(* IEC 61131-3 sources: HMITools/src/Ar/HMITools, 32 files *)

(* ---- EditorControl.typ ---- *)
(*
* File: EditorControl.typ
* Copyright (c) 2023 Loupe
* https://loupe.team
*
* This file is part of HMITools, licensed under the MIT License.
*
*)
(*Application Editor*)

TYPE
	HMI_Editor_Controller_typ : 	STRUCT
		CMD : HMI_Editor_Controller_CMD_typ;
		HMI : HMI_EditControl_typ;
		Internal : HMI_Editor_Controller_int_typ;
	END_STRUCT;
	HMI_Editor_Controller_int_typ : 	STRUCT
		CMD : HMI_Editor_Controller_CMD_typ;
	END_STRUCT;
	HMI_Editor_Controller_CMD_typ : 	STRUCT
		Load : BOOL;
		Save : BOOL;
		Clear : BOOL;
	END_STRUCT;
END_TYPE

(*HMI Connections*)

TYPE
	HMI_EditControl_Internal_typ : 	STRUCT
		CurrentLineText : STRING[200];
		CurrentLineIndex : UINT;
		CommandState : USINT;
		EditText : STRING[80];
		DesiredLine : USINT;
		DesiredColumn : USINT;
		Offset : USINT;
		Count : USINT;
		highlightmode : USINT;
	END_STRUCT;
	HMI_EditControl_Runtime_Edit_typ : 	STRUCT
		CursorLineDp : UINT;
		CursorColumnDp : UINT;
		InsertModeDp : UINT;
		ModifiedDp : UINT;
		SelectionModeDp : UINT;
	END_STRUCT;
	HMI_EditControl_Runtime_Comp_typ : 	STRUCT
		CompletionDP : UINT;
	END_STRUCT;
	HMI_EditControl_Runtime_Cmds_typ : 	STRUCT
		ResponseDp : STRING[80];
		RequestDp : STRING[80];
		StatusDP : UINT;
	END_STRUCT;
	HMI_EditControl_Runtime_typ : 	STRUCT
		StatusDp : UINT;
		BusyDp : UINT;
		Commands : HMI_EditControl_Runtime_Cmds_typ;
		Completion : HMI_EditControl_Runtime_Comp_typ;
		Edit : HMI_EditControl_Runtime_Edit_typ;
	END_STRUCT;
	HMI_EditControl_Value_typ : 	STRUCT
		Content : STRING[1000];
		URLDp : STRING[80];
	END_STRUCT;
	HMI_EditControl_typ : 	STRUCT
		Value : HMI_EditControl_Value_typ;
		Runtime : HMI_EditControl_Runtime_typ;
		internal : HMI_EditControl_Internal_typ;
		Command : HMI_EditControl_CMDS;
	END_STRUCT;
	HMI_EditControl_CMDS :
		(
		EC_,
		EC_APPEND,
		EC_CLEAR,
		EC_DELETE,
		EC_GET_LINE,
		EC_GET_MARKED_TEXT,
		EC_GET_TEXT_SIZE,
		EC_GOTO,
		EC_HIGHLIGHT,
		EC_INSERT,
		EC_LOAD,
		EC_READ,
		EC_REPLACE_MARKED_TEXT,
		EC_SAVE,
		EC_UPDATE
		);
END_TYPE

(* ---- HMI_Basic.typ ---- *)
(*
* File: HMI_Basic.typ
* Copyright (c) 2023 Loupe
* https://loupe.team
*
* This file is part of HMITools, licensed under the MIT License.
*
*)

TYPE
	HMI_StatusBits_enum :
		(
		HMI_STATBIT_VIS := 0,
		HMI_STATBIT_LOCK,
		HMI_STATBIT_FOCUS,
		HMI_STATBIT_TOUCHPAD
		);
	HMI_Layer_typ : 	STRUCT
		StatusDP : UINT;
	END_STRUCT;
	HMI_Shape_typ : 	STRUCT
		StatusDP : UINT;
		ColorDP : UINT;
	END_STRUCT;
	HMI_Scale_typ : 	STRUCT
		Value : REAL;
		MinDP : REAL;
		MaxDP : REAL;
		RangeStartDP : REAL;
		RangeEndDP : REAL;
		RangeColorDP : UINT;
		StatusDP : UINT;
		ColorDP : UINT;
	END_STRUCT;
	HMI_Listbox_typ : 	STRUCT
		IndexDP : DINT;
		MinDP : UINT;
		MaxDP : UINT;
		OptionDP : UINT;
		StatusDP : UINT;
		ColorDP : UINT;
		CompletionDP : UINT;
		PageSize : UINT;
	END_STRUCT;
	HMI_Bitmap_typ : 	STRUCT
		IndexDP : UINT;
		StatusDP : UINT;
	END_STRUCT;
	HMI_StringIn_typ : 	STRUCT
		String : STRING[HMI_STRLEN_IN];
		StatusDP : UINT;
		ColorDP : UINT;
		CompletionDP : UINT;
	END_STRUCT;
	HMI_Dropdown_typ : 	STRUCT
		IndexDP : UINT;
		StatusDP : UINT;
		ColorDP : UINT;
	END_STRUCT;
	HMI_TextBox_typ : 	STRUCT
		IndexDP : UINT;
		StatusDP : UINT;
		ColorDP : UINT;
	END_STRUCT;
	HMI_NumericIn_typ : 	STRUCT
		Value : REAL;
		MinDP : REAL;
		MaxDP : REAL;
		StatusDP : UINT;
		ColorDP : UINT;
		CompletionDP : UINT;
	END_STRUCT;
	HMI_NumericOut_typ : 	STRUCT
		Value : REAL;
		StatusDP : UINT;
		ColorDP : UINT;
	END_STRUCT;
	HMI_ButtonVC3_typ : 	STRUCT
		CMD : USINT;
		Lock : UINT;
		ColorDP : UINT;
		LEDDP : USINT;
	END_STRUCT;
	HMI_Button_typ : 	STRUCT
		CMD : BOOL;
		Confirm : BOOL;
		StatusDP : UINT;
		IndexDP : UINT;
		ColorDP : UINT;
		LEDDP : USINT;
	END_STRUCT;
	HMI_SecondaryTab_typ : 	STRUCT
		ChangeToSecondaryTab : BOOL; (*CMD to change to this secondary tab*)
		PageIndex : UINT; (*Page index for this secondary tab*)
	END_STRUCT;
	HMI_PrimaryTab_typ : 	STRUCT
		CurrentSecondaryTab : UINT; (*Current secondary tab*)
		ChangeToPrimaryTab : BOOL; (*CMD to change to this primary tab*)
		Group : UINT; (*Group to which the primary tab belongs*)
		SecondaryTabArray : ARRAY[0..HMI_MAI_TABS]OF HMI_SecondaryTab_typ; (*Array of secondary tabs*)
	END_STRUCT;
	HMI_Tabs_typ : 	STRUCT
		CurrentPrimaryTab : UINT;
		PrimaryTabArray : ARRAY[0..HMI_MAI_TABS]OF HMI_PrimaryTab_typ;
	END_STRUCT;
	HMI_Basic_typ : 	STRUCT
		PageChangeDP : UINT;
		PageCurrentDP : UINT;
		LanguageChangeDP : UINT;
		LanguageCurrentDP : UINT;
		ScreensaverDP : UINT;
		ScreensaverTimeDP : UINT;
		BacklightDP : UINT;
		BacklightTimeDP : UINT;
		CalibrationStateDP : UINT;
		VCHandle : UDINT;
		Tabs : HMI_Tabs_typ;
	END_STRUCT;
END_TYPE

(* ---- HMI_File_Browse.typ ---- *)
(*
* File: HMI_File_Browse.typ
* Copyright (c) 2023 Loupe
* https://loupe.team
*
* This file is part of HMITools, licensed under the MIT License.
*
*)

TYPE
	HMI_File_Browse_internal_typ : 	STRUCT
		TempFileList : UDINT;
		TempFileSelection : STRING[LIST_BOX_STRING_SIZE];
		oldFileIndex : DINT;
		oldFileSelection : STRING[LIST_BOX_STRING_SIZE];
		NameFilter : STRING[LIST_BOX_STRING_SIZE];
		PathStrSize : UINT;
		InternalBrowsingPath : STRING[LIST_BOX_STRING_SIZE];
		i : UINT;
		IsolatedChar : USINT;
		FileNameSelector : ListBoxFub;
		FileExtensionSelector : ListBoxFub;
		Directory : DirectoryFub;
		TON_0 : TON;
	END_STRUCT;
END_TYPE

(* ---- HMI_Trend.typ ---- *)
(*
* File: HMI_Trend.typ
* Copyright (c) 2023 Loupe
* https://loupe.team
*
* This file is part of HMITools, licensed under the MIT License.
*
*)

TYPE
	HMI_TrendValueScale_typ : 	STRUCT
		ColorDP : UINT;
		ScrollManual : REAL;
		ZoomManual : REAL;
		ZoomScroll : Trend_ZoomScroll;
		StatusDP : UINT;
	END_STRUCT;
	HMI_TrendTimeContainer_typ : 	STRUCT
		ColorDP : UINT;
		CursorTimeDP : ARRAY[0..HMI_TREND_MAI_CURSOR]OF REAL; (*Time at the current Trend.CursorPositionDP.*)
		ZoomManual : REAL;
		ScrollManual : REAL;
		ModeManual : UINT;
		ZoomScroll : Trend_ZoomScroll;
		StatusDP : UINT;
	END_STRUCT;
	HMI_TrendScaleContainer_typ : 	STRUCT
		ColorDP : UINT;
		StatusDP : UINT;
	END_STRUCT;
	HMI_TrendCurve_typ : 	STRUCT
		ColorDP : UINT;
		CursorValueDP : ARRAY[0..HMI_TREND_MAI_CURSOR]OF REAL; (*Value of the current curve data at the current Trend.CursorPositionDP.*)
		StatusDP : UINT;
	END_STRUCT;
	HMI_TrendGrid_typ : 	STRUCT
		ColorDP : UINT;
		StatusDP : UINT;
	END_STRUCT;
	HMI_Trend_typ : 	STRUCT
		ColorDP : UINT; (*ColorDP should be mapped to the ColorDatapoint in the Trend object on the page.*)
		SelectItemDP : UINT; (*SelectItemDP should be mapped to the SelectItemDatapoint in the Trend object on the page.*)
		StatusDP : UINT; (*StatusDP should be mapped to the StatusDatapoint in the Trend object on the page.*)
		CursorPositionDP : ARRAY[0..HMI_TREND_MAI_CURSOR]OF REAL; (*CursorPositionDP should be mapped to the Cursor PositionDatapoint in the Trend object in the trend editor.
This is used to set the current position of the cursor, as a percentage within full range.*)
		CursorStatusDP : ARRAY[0..HMI_TREND_MAI_CURSOR]OF UINT; (*CursorStatusDP should be mapped to the Cursor StatusDatapoint in the Trend object in the trend editor.*)
		Grid : HMI_TrendGrid_typ; (*Grid variables should be mapped to the TrendGrid in the trend editor.*)
		Curve : ARRAY[0..HMI_TREND_MAI_CURVE]OF HMI_TrendCurve_typ; (*Curve variables should be mapped to the TrendCurve objects in the trend editor.*)
		ScaleContainer : ARRAY[0..HMI_TREND_MAI_SCALECONTAINER]OF HMI_TrendScaleContainer_typ; (*ScaleContainer variables should be mapped to the TrendScaleContainer objects in the trend editor.*)
		TimeContainer : HMI_TrendTimeContainer_typ; (*TimeContainer variables should be mapped to the TrendTimeContainer object in the trend editor.*)
		ValueScale : ARRAY[0..HMI_TREND_MAI_VALUESCALE]OF HMI_TrendValueScale_typ; (*ValueScale variables should be mapped to the TrendValueScale objects in the trend editor.*)
		GlobalXZoomManual : REAL; (*Global zoom and scroll datapoints can be mapped to the zoom and scroll datapoints of ALL TrendTimeContainer and TrendValueScale objects in the trend editor.
This allows for one command to affect the ENTIRE trend.
Local zoom and scroll datapoints in the Trend.TimeContainer and Trend.ValueScale structures can be used to perform zooming and scrolling independently for each TrendTimeContainer and TrendValueScale object.
For manual operation, use the manual datapoints. For automatic operation, use the respective ZoomScroll FUB instance.*)
		GlobalXScrollManual : REAL;
		GlobalXScrollModeManual : UINT;
		GlobalXZoomScroll : Trend_ZoomScroll;
		GlobalYScrollManual : REAL;
		GlobalYZoomManual : REAL;
		GlobalYZoomScroll : Trend_ZoomScroll;
	END_STRUCT;
END_TYPE

(* ---- HMITools.typ ---- *)
(*
* File: HMITools.typ
* Copyright (c) 2023 Loupe
* https://loupe.team
*
* This file is part of HMITools, licensed under the MIT License.
*
*)

TYPE
	HMI_ERR_enum :
		(
		HMI_ERR_OK := 0,
		HMI_ERR_INVALIDINPUT := 50000,
		HMI_ERR_BUSY := 65535
		);
END_TYPE

(* ---- LogViewer.typ ---- *)
(*
* File: LogViewer.typ
* Copyright (c) 2023 Loupe
* https://loupe.team
*
* This file is part of HMITools, licensed under the MIT License.
*
*)

TYPE
	LogView_HMI_typ : 	STRUCT
		ListBox : HMI_Listbox_typ;
		GoToTopButton : HMI_Button_typ;
		PageUpButton : HMI_Button_typ;
		PageDownButton : HMI_Button_typ;
		UpButton : HMI_Button_typ;
		DownButton : HMI_Button_typ;
		Text : STRING[LIST_BOX_STRING_SIZE];
		FilterString : STRING[80];
		MaxAlarms : UDINT;
		AlarmList : UDINT;
		internal : LogView_HMI_internal_typ;
	END_STRUCT;
	LogView_HMI_internal_typ : 	STRUCT
		Offset : DINT;
		SelectedAlarmIndex : UDINT;
		SelectedListIndex : UINT;
		oSelectedListIndex : UINT;
		NumberAlarms : UINT;
	END_STRUCT;
	LogView_typ : 	STRUCT
		IN : LogView_IN_typ;
		OUT : LogView_OUT_typ;
		Internal : LogView_Internal_typ;
	END_STRUCT;
	LogView_IN_typ : 	STRUCT  (*Logger Variables*)
		PAR : LogView_PAR_typ;
		CMD : LogView_CMD_typ;
		CFG : LogView_CFG_typ;
	END_STRUCT;
	LogView_PAR_typ : 	STRUCT  (*Logger Variables*)
		LoggerName : STRING[80];
		Offset : DINT;
	END_STRUCT;
	LogView_CMD_typ : 	STRUCT  (*Logger Variables*)
		GoToTop : BOOL;
	END_STRUCT;
	LogView_CFG_typ : 	STRUCT  (*Logger Variables*)
		MaxLogs : UINT;
	END_STRUCT;
	LogView_OUT_typ : 	STRUCT  (*Logger Variables*)
		STAT : LogView_STAT_typ;
		NumberAlarms : UDINT;
	END_STRUCT;
	LogView_STAT_typ : 	STRUCT  (*Logger Variables*)
		Done : BOOL;
		Busy : BOOL;
		Error : BOOL;
		ErrorID : DINT;
		ErrorString : STRING[80];
	END_STRUCT;
	LogView_Internal_typ : 	STRUCT  (*Logger Variables*)
		GetIdent: ArEventLogGetIdent;
		GetRecordID: ArEventLogGetLatestRecordID;
		GetTopAlarm : LogView_GetAlarm;
		GetBottomAlarm : LogView_GetAlarm;
		Buffer : Buffer_typ;
		OffsetIndex : UDINT;
		LoggerName : STRING[80];
		Ident : UDINT;
	END_STRUCT;
	ArEventLogREAD: 	STRUCT  (*Header data for log entry*)
		lenAscii : UDINT; (*Length of the ASCII log data*)
		errornr : UDINT; (*Error number of the entry*)
		errTime : DTStructure;
	END_STRUCT;
	LogView_GetAlarm : 	STRUCT
		ReadItem : ArEventLogRead; (*ArEventLog: ArEventLogRead FUB*)
		ReadAddData: ArEventLogReadAddData; (*For reading the message text*)
		ReadData : ArEventLogREAD;
		convertUTC : UtcDT_TO_LocalDTStructure;
		BinaryData : ARRAY[0..255]OF USINT;
		ASCIIData : ARRAY[0..255]OF USINT;
	END_STRUCT;
	LogData : 	STRUCT
		String : STRING[LIST_BOX_STRING_SIZE];
		Index : UDINT;
	END_STRUCT;
END_TYPE

(* ---- RecipeMgr.typ ---- *)
(*
* File: RecipeMgr.typ
* Copyright (c) 2023 Loupe
* https://loupe.team
*
* This file is part of HMITools, licensed under the MIT License.
*
*)

TYPE
	RecMgr_HMI_typ : 	STRUCT
		RetrieveFromSystem : HMI_Button_typ; (*Retrieve current system recipe (copy from pSystemRecipe to pHMIRecipe)*)
		ApplyToSystem : HMI_Button_typ; (*Apply current recipe to system (copy from pHMIRecipe to pSystemRecipe)*)
		Modified : HMI_Bitmap_typ;
	END_STRUCT;
	RecMgr_IN_typ : 	STRUCT
		pHMIRecipe : UDINT; (*HMI Recipe location. Given as an address.*)
		pSystemRecipe : UDINT; (*System Recipe location. Given as an address.*)
		RecipeLength : UDINT; (*Size of the recipe in bytes*)
		LoggerName : STRING[LOG_STRLEN_LOGGERNAME];
	END_STRUCT;
	RecipeMgr_typ : 	STRUCT
		IN : RecMgr_IN_typ;
		HMI : RecMgr_HMI_typ;
	END_STRUCT;
END_TYPE

(* ---- Updater.typ ---- *)
(*
* File: Updater.typ
* Copyright (c) 2023 Loupe
* https://loupe.team
*
* This file is part of HMITools, licensed under the MIT License.
*
*)

TYPE
	RecipeUpdater_Internal_typ : 	STRUCT
		State : RecipeUpdater_STATE;
		DirRead : DirRead;
		CurrentFile : fiDIR_READ_DATA;
	END_STRUCT;
	RecipeUpdater_STATE :
		(
		RecipeUpdater_ST_IDLE,
		RecipeUpdater_ST_ReadDirectory,
		RecipeUpdater_ST_ReadFile,
		RecipeUpdater_ST_WAIT,
		RecipeUpdater_ST_UpdateFile,
		RecipeUpdater_ST_Done,
		RecipeUpdater_ST_
		);
END_TYPE

(* ---- CustomControl.st ---- *)
(*
* File: CustomControl.st
* Copyright (c) 2023 Loupe
* https://loupe.team
*
* This file is part of HMITools, licensed under the MIT License.
*
*)

(* TODO: Add your comment here *)
FUNCTION ControlTouch

	ControlTouch:=0;

	State:= BOOL_TO_UINT(StatusDP.4)+BOOL_TO_UINT(StatusDP.5)*2;

	CASE State OF

		0:
			StatusDP.1:=1;
			IF StatusDP.13 = 1 THEN
				StatusDP.13:=0;
				//set state
				StatusDP.4:=1;
			END_IF
		1:
			StatusDP.1:=1;
			ControlTouch:=1;

			IF StatusDP.13 = 1 THEN
				StatusDP.13:=0;
				StatusDP.1:=0;
				//set state
				StatusDP.4:=0;
				StatusDP.5:=1;
				StatusDP.3:=1;
			END_IF

		2:
			IF StatusDP.12 = 1 THEN
				StatusDP.4:=1;
				StatusDP.5:=1;
			END_IF

		3:
			IF StatusDP.12 = 0 THEN
				StatusDP.4:=0;
				StatusDP.5:=0;
			END_IF

	END_CASE

END_FUNCTION

FUNCTION ControlDismiss

	ControlDismiss:=0;

	StatusDP.4:=0;
	StatusDP.5:=0;

END_FUNCTION

(* ---- Editor_fn.st ---- *)
(*
* File: Editor_fn.st
* Copyright (c) 2023 Loupe
* https://loupe.team
*
* This file is part of HMITools, licensed under the MIT License.
*
*)

(* TODO: Add your comment here *)
FUNCTION Editor_fn

	Editor_fn:=0;

	IF EditorController.CMD.Save THEN
		EditorController.HMI.Command:= EC_SAVE;
		EditorController.Internal.CMD.Save:=1;
	ELSIF EditorController.CMD.Load THEN
		EditorController.HMI.Command:= EC_LOAD;
		EditorController.Internal.CMD.Load:=1;
	ELSIF EditorController.CMD.Clear THEN
		EditorController.HMI.Command:= EC_CLEAR;
		EditorController.Internal.CMD.Clear:=1;
	END_IF

	IF NOT EditorController.CMD.Save THEN
		EditorController.Internal.CMD.Save:=0;
	ELSIF NOT EditorController.CMD.Load THEN
		EditorController.Internal.CMD.Load:=0;
	ELSIF NOT EditorController.CMD.Clear THEN
		EditorController.Internal.CMD.Clear:=0;
	END_IF

	EditorControl(EditorController.HMI);

END_FUNCTION

(* Controls an HMI edit control *)
FUNCTION EditorControl

	EditorControl:=0;

	CASE Editor.internal.CommandState OF
		0:
			Editor.internal.CommandState:=Editor.internal.CommandState+1;

			CASE Editor.Command OF
				EC_APPEND://append
					EditControl_CS_append(Editor.internal.EditText,Editor.Runtime.Commands.RequestDp);
				EC_CLEAR://clear
					Editor.Runtime.Commands.RequestDp:='clear';
				EC_DELETE://delete
					Editor.Runtime.Commands.RequestDp:='delete';
				EC_GET_LINE://getline
					EditControl_CS_getline(Editor.internal.CurrentLineIndex,Editor.Runtime.Commands.RequestDp);
				EC_GET_MARKED_TEXT://getmarkedtext
					Editor.Runtime.Commands.RequestDp:='getmarkedtext';
				EC_GET_TEXT_SIZE://gettextsize
					Editor.Runtime.Commands.RequestDp:='gettextsize';
				EC_GOTO://goto
					EditControl_CS_goto(Editor.internal.DesiredLine,Editor.internal.DesiredColumn,Editor.Runtime.Commands.RequestDp);
				EC_HIGHLIGHT://highlight
					EditControl_CS_highlight(Editor.internal.DesiredLine,Editor.internal.highlightmode,Editor.Runtime.Commands.RequestDp);
				EC_INSERT://insert
					EditControl_CS_insert(Editor.internal.EditText,Editor.internal.DesiredLine,Editor.Runtime.Commands.RequestDp);
				EC_LOAD://load
					Editor.Runtime.Commands.RequestDp:='load';
				EC_READ://read
					EditControl_CS_read(Editor.internal.Offset,Editor.internal.Count,Editor.Runtime.Commands.RequestDp);
				EC_REPLACE_MARKED_TEXT://replacemarkedtext
					EditControl_CS_replacemarked(Editor.internal.EditText,Editor.Runtime.Commands.RequestDp);
				EC_SAVE://save
					Editor.Runtime.Commands.RequestDp:='save';
				EC_UPDATE://update
					Editor.Runtime.Commands.RequestDp:='update';
				ELSE
					Editor.internal.CommandState:=0;
			END_CASE

		1:
			IF Editor.Runtime.Commands.StatusDP = 0 THEN
				Editor.internal.CommandState:=Editor.internal.CommandState+1;
			END_IF

		2:
			Editor.Command:=0;
			Editor.Runtime.Commands.StatusDP:=	1;
			Editor.internal.CommandState:=Editor.internal.CommandState+1;

		3:
			IF Editor.Runtime.Commands.StatusDP = 0 THEN
				Editor.internal.CurrentLineText:=Editor.Runtime.Commands.ResponseDp;
				Editor.internal.CommandState:=0;
			END_IF
	END_CASE;

END_FUNCTION

FUNCTION EditControl_CS_append

	EditControl_CS_append:=0;

	Output:=CONCAT('append text=',Text);

END_FUNCTION

FUNCTION EditControl_CS_getline

	EditControl_CS_getline:=0;

	brsitoa(Line,ADR(temp));
	Output:=CONCAT('getline line=',temp);

END_FUNCTION

FUNCTION EditControl_CS_goto

	EditControl_CS_goto:=0;

	brsitoa(Col,ADR(temp));
	Output:=CONCAT('goto col=',temp);
	Output:=CONCAT(Output,' line=');
	brsitoa(Line,ADR(temp));
	Output:=CONCAT(Output,temp);

END_FUNCTION

FUNCTION EditControl_CS_highlight

	EditControl_CS_highlight:=0;

	brsitoa(Value,ADR(temp));
	IF Mode = 0 THEN
		Output:=CONCAT('highlight offset=',temp);
	ELSE
		Output:=CONCAT('highlight line=',temp);
	END_IF
END_FUNCTION

FUNCTION EditControl_CS_insert

	EditControl_CS_insert:=0;

	brsitoa(Line,ADR(temp));
	Output:=CONCAT('insert line=',temp);
	Output:=CONCAT(Output,' text=');
	Output:=CONCAT(Output,Text);
END_FUNCTION

FUNCTION EditControl_CS_read

	EditControl_CS_read:=0;

	brsitoa(Offset,ADR(temp));
	Output:=CONCAT('read offset=',temp);
	Output:=CONCAT(Output,' count=');
	brsitoa(Count,ADR(temp));
	Output:=CONCAT(Output,temp);

END_FUNCTION

FUNCTION EditControl_CS_replacemarked

	EditControl_CS_replacemarked:=0;

	Output:=CONCAT('replacemarkedtext text=',Text);

END_FUNCTION

FUNCTION EditControl_CS_replaceline

	EditControl_CS_replaceline:=0;

	brsitoa(Line,ADR(temp));
	Output:=CONCAT('update line=',temp);
	Output:=CONCAT(Output,' text=');
	Output:=CONCAT(Output,Text);

END_FUNCTION

(* ---- GetDataObjectList.st ---- *)
(*
* File: GetDataObjectList.st
* Copyright (c) 2023 Loupe
* https://loupe.team
*
* This file is part of HMITools, licensed under the MIT License.
*
*)
(*  *)
FUNCTION GetDataObjectList

		//Keep track of the objects that we've gone through
	//unsigned int objectIndex = 0;
	objectIndex:= 0;

	//Number of variables that have been found
	numberVariables:=0;
	duplicate:=0;
	index:=0;

	//Check for valid inputs
	IF( List = 0 ) THEN
		GetDataObjectList:=0;
		RETURN;
	END_IF

	//Clear out any bad data
	Files ACCESS List;
	brsmemset(ADR(Files ),0,MaxObjects*(LIST_BOX_STRING_SIZE+1));

	//Look through all the objects
	WHILE( MO_list(objectIndex, ADR(objectIndex), ADR(Item)) = 0 AND numberVariables < MaxObjects)DO
		//If it is a cyclic object check if it has the variable
		duplicate:=0;
		IF( Item.type = 16#41) THEN
			FOR index:= 0 TO numberVariables DO
				IF(brsstrcmp(ADR(Item.name),ADR(Files[index]))=0)THEN
					duplicate:=1;
					EXIT;
				END_IF
			END_FOR
			IF(NOT duplicate) THEN
				brsstrcpy( ADR(Files[numberVariables]),ADR(Item.name));
				numberVariables:=numberVariables+1;
			END_IF
		END_IF
	END_WHILE

	//Return the number of found variables to make it easy to add to the list outside the function.
	GetDataObjectList:= numberVariables;

END_FUNCTION

(* ---- HMI_FindCurrentTab.st ---- *)
(*
* File: HMI_FindCurrentTab.st
* Copyright (c) 2023 Loupe
* https://loupe.team
*
* This file is part of HMITools, licensed under the MIT License.
*
*)

(****************************************************************************************)
(* Function to find the current primary and secondary tab based on the current page 	*)
(****************************************************************************************)

(* Setting CurrentPrimaryTab		DONE and TESTED DFB 20110519 *)
(* Setting CurrentSecondaryTab		DONE and TESTED DFB 20110519 *)

FUNCTION HMI_FindCurrentTab

(****************************************************)
(* Set return value to get rid of compile warning 	*)
(****************************************************)

HMI_FindCurrentTab:=	FALSE;

(* Loop through primary and secondary tabs.
	If the current page matches a secondary page,
	set the secondary tab accordingly.
	If a match is not found, do nothing. *)

(* 0 IS NOT A VALID TAB PAGE INDEX *)

FOR p:=0 TO HMI_MAI_TABS BY 1 DO

	FOR ss:=0 TO HMI_MAI_TABS BY 1 DO

		IF( 	(t.PageCurrentDP = t.Tabs.PrimaryTabArray[p].SecondaryTabArray[ss].PageIndex)
			AND	(t.Tabs.PrimaryTabArray[p].SecondaryTabArray[ss].PageIndex <> 0)
   			)THEN

			t.Tabs.CurrentPrimaryTab:=	p;

			t.Tabs.PrimaryTabArray[p].CurrentSecondaryTab:=	ss;

			RETURN;

		END_IF

	END_FOR

END_FOR

END_FUNCTION

(* ---- HMI_Hide.st ---- *)
(*
* File: HMI_Hide.st
* Copyright (c) 2023 Loupe
* https://loupe.team
*
* This file is part of HMITools, licensed under the MIT License.
*
*)

(****************************************************************)
(* Hide an item on the screen 									*)
(****************************************************************)

(* Function			DONE and TESTED DFB 20110503 *)

FUNCTION HMI_Hide

(****************************************************************)
(* Set return value to get rid of compiler error				*)
(****************************************************************)

HMI_Hide:=	FALSE;

(****************************************************************)
(* Set/clear proper bit in StatusDP								*)
(****************************************************************)

StatusDP.HMI_STATBIT_VIS:=	HMI_INVISIBLE;

END_FUNCTION

(* ---- HMI_Lock.st ---- *)
(*
* File: HMI_Lock.st
* Copyright (c) 2023 Loupe
* https://loupe.team
*
* This file is part of HMITools, licensed under the MIT License.
*
*)

(****************************************************************)
(* Lock an item on the screen 									*)
(****************************************************************)

(* Function			DONE and TESTED DFB 20110503 *)

FUNCTION HMI_Lock

(****************************************************************)
(* Set return value to get rid of compiler error				*)
(****************************************************************)

HMI_Lock:=	FALSE;

(****************************************************************)
(* Set/clear proper bit in StatusDP								*)
(****************************************************************)

StatusDP.HMI_STATBIT_LOCK:=	HMI_LOCKED;

END_FUNCTION

(* ---- HMI_OpenTouchpad.st ---- *)
(*
* File: HMI_OpenTouchpad.st
* Copyright (c) 2023 Loupe
* https://loupe.team
*
* This file is part of HMITools, licensed under the MIT License.
*
*)

(********************************************************************)
(* Opens the touchpad for an item on the screen 					*)
(********************************************************************)

(* Function			DONE and TESTED DFB 20110504 *)

FUNCTION HMI_OpenTouchpad

(****************************************************************)
(* Set return value to get rid of compiler error				*)
(****************************************************************)

HMI_OpenTouchpad:=	FALSE;

(****************************************************************)
(* Set/clear proper bit in StatusDP								*)
(****************************************************************)

StatusDP.HMI_STATBIT_TOUCHPAD:=	1;

END_FUNCTION

(* ---- HMI_ResetFocus.st ---- *)
(*
* File: HMI_ResetFocus.st
* Copyright (c) 2023 Loupe
* https://loupe.team
*
* This file is part of HMITools, licensed under the MIT License.
*
*)

(************************************************************************************)
(* Resets the focus bit for an item on the screen. THIS DOES NOT MOVE THE FOCUS!	*)
(************************************************************************************)

(* Function			DONE and TESTED DFB 20110504 *)

FUNCTION HMI_ResetFocus

(****************************************************************)
(* Set return value to get rid of compiler error				*)
(****************************************************************)

HMI_ResetFocus:=	FALSE;

(****************************************************************)
(* Set/clear proper bit in StatusDP								*)
(****************************************************************)

StatusDP.HMI_STATBIT_FOCUS:=	0;

END_FUNCTION

(* ---- HMI_SetFocus.st ---- *)
(*
* File: HMI_SetFocus.st
* Copyright (c) 2023 Loupe
* https://loupe.team
*
* This file is part of HMITools, licensed under the MIT License.
*
*)

(********************************************************************)
(* Sets the focus for an item on the screen. FOCUS MUST BE RESET!	*)
(********************************************************************)

(* Function			DONE and TESTED DFB 20110504 *)

FUNCTION HMI_SetFocus

(****************************************************************)
(* Set return value to get rid of compiler error				*)
(****************************************************************)

HMI_SetFocus:=	FALSE;

(****************************************************************)
(* Set/clear proper bit in StatusDP								*)
(****************************************************************)

StatusDP.HMI_STATBIT_FOCUS:=	1;

END_FUNCTION

(* ---- HMI_Show.st ---- *)
(*
* File: HMI_Show.st
* Copyright (c) 2023 Loupe
* https://loupe.team
*
* This file is part of HMITools, licensed under the MIT License.
*
*)

(****************************************************************)
(* Show an item on the screen 									*)
(****************************************************************)

(* Function			DONE and TESTED DFB 20110503 *)

FUNCTION HMI_Show

(****************************************************************)
(* Set return value to get rid of compiler error				*)
(****************************************************************)

HMI_Show:=	FALSE;

(****************************************************************)
(* Set/clear proper bit in StatusDP								*)
(****************************************************************)

StatusDP.HMI_STATBIT_VIS:=	HMI_VISIBLE;

END_FUNCTION

(* ---- HMI_TabControlFn_Cyclic.st ---- *)
(*
* File: HMI_TabControlFn_Cyclic.st
* Copyright (c) 2023 Loupe
* https://loupe.team
*
* This file is part of HMITools, licensed under the MIT License.
*
*)

(********************************************************************)
(* Handle tab based page switching 									*)
(********************************************************************)

(* Finding current tab						see HMI_FindCurrentTab.st *)

(* Primary tab changes						DONE and TESTED DFB 20110729 *)
	(* Changing within a group				DONE and TESTED DFB 20110729 *)
	(* Changing outside a group				DONE and TESTED DFB 20110729 *)
		(* From group to no group			DONE and TESTED DFB 20110729 *)
		(* From no group to group			DONE and TESTED DFB 20110729 *)
		(* From no group to no group		DONE and TESTED DFB 20110729 *)
	(* PageIndex = 0						DONE and TESTED DFB 20110729 *)

(* Secondary tab changes					DONE and TESTED DFB 20110729 *)

(* Clearing inappropriate SecondaryTabs		DONE and TESTED DFB 20110729 *)

(* Checking for no tabs active				DONE and TESTED DFB 20110729 *)
	(* Primary								DONE and TESTED DFB 20110729 *)
	(* Secondary							DONE and TESTED DFB 20110729 *)

(* Implementation with HMI					DONE and TESTED DFB 20110801 *)

(* Allowing external page changes			DONE and TESTED DFB 20110801 *)

FUNCTION HMI_TabControlFn_Cyclic

(********************************************************************************)
(* NOTE: THIS FUNCTION MUST RUN IN CYCLIC 8 WITH A CYCLE TIME < ~50ms			*)
(********************************************************************************)

(****************************************************)
(* Set return value to get rid of compile warning 	*)
(****************************************************)

HMI_TabControlFn_Cyclic:=	FALSE;

(****************************************************)
(* Find the current tab 							*)
(****************************************************)

HMI_FindCurrentTab( t );

(****************************************************)
(* Handle external page changes						*)
(****************************************************)

(* Check for ChangePage active *)

IF( 	(t.PageChangeDP <> 65535)
	AND	(t.PageChangeDP <> 0)
 	)THEN

	(* If ChangePage is active, then reset
		Current tab CMDs and do not execute rest of fn *)

	t.Tabs.PrimaryTabArray[t.Tabs.CurrentPrimaryTab].ChangeToPrimaryTab:=	0;

	t.Tabs.PrimaryTabArray[t.Tabs.CurrentPrimaryTab]
			.SecondaryTabArray[t.Tabs.PrimaryTabArray[t.Tabs.CurrentPrimaryTab].CurrentSecondaryTab]
			.ChangeToSecondaryTab:=	0;

	RETURN;

END_IF

(****************************************************)
(* Handle primary tab page changes 					*)
(****************************************************)

FOR p:=0 TO HMI_MAI_TABS BY 1 DO

	(* Do not check the CurrentPrimaryTab *)

	IF( p <> t.Tabs.CurrentPrimaryTab )THEN

		(* If a NEW primary tab is chosen, then reset current primary tab and change page *)

		IF( t.Tabs.PrimaryTabArray[p].ChangeToPrimaryTab )THEN

			//t.Tabs.PrimaryTabArray[p].ChangeToPrimaryTab:=	0;

			(* If desired tab (p) is in a group, and you are in that group,
				change to the CurrentPrimaryTab's CurrentSecondaryTab *)

			IF( 	(t.Tabs.PrimaryTabArray[p].Group <> 0)
				AND	(t.Tabs.PrimaryTabArray[p].Group = t.Tabs.PrimaryTabArray[t.Tabs.CurrentPrimaryTab].Group)
				)THEN

				SecondaryTabIndex:=	t.Tabs.PrimaryTabArray[t.Tabs.CurrentPrimaryTab].CurrentSecondaryTab;

			(* Otherwise, change to the desired primary tab's (p) CurrentSecondaryTab *)

			ELSE

				SecondaryTabIndex:=	t.Tabs.PrimaryTabArray[p].CurrentSecondaryTab;

			END_IF

			(* Change to the correct secondary tab if it has a valid PageIndex and you are not already there *)

			IF( 	(t.Tabs.PrimaryTabArray[p].SecondaryTabArray[SecondaryTabIndex].PageIndex <> 0)
				AND	(t.Tabs.PrimaryTabArray[p].SecondaryTabArray[SecondaryTabIndex].PageIndex <> t.PageCurrentDP)
				)THEN

				(* Change Page and set Tab CMDs accordingly *)

				t.PageChangeDP:=
					t.Tabs.PrimaryTabArray[p].SecondaryTabArray[SecondaryTabIndex].PageIndex;

				(* Set current secondary tab *)

				t.Tabs.PrimaryTabArray[p]
						.SecondaryTabArray[SecondaryTabIndex]
						.ChangeToSecondaryTab:=	1;

				(* Reset previous primary and secondary tab *)

				t.Tabs.PrimaryTabArray[t.Tabs.CurrentPrimaryTab].ChangeToPrimaryTab:=	0;

				t.Tabs.PrimaryTabArray[t.Tabs.CurrentPrimaryTab]
						.SecondaryTabArray[t.Tabs.PrimaryTabArray[t.Tabs.CurrentPrimaryTab].CurrentSecondaryTab]
						.ChangeToSecondaryTab:=	0;

			ELSE

				(* Error - Reset CMD and do nothing *)

				t.Tabs.PrimaryTabArray[p].ChangeToPrimaryTab:=	0;

			END_IF // ChangePage

			RETURN;

		END_IF // ChangeToPrimaryTab

	END_IF // Not CurrentPrimaryTab

END_FOR

(****************************************************)
(* Handle secondary tab page changes 				*)
(****************************************************)

(* Loop through CurrentPrimaryTab's secondary tabs to look for commands *)

FOR ss:=0 TO HMI_MAI_TABS BY 1 DO

	(* Do not check the current secondary tab *)

	IF( ss <> t.Tabs.PrimaryTabArray[t.Tabs.CurrentPrimaryTab].CurrentSecondaryTab )THEN

		(* If a NEW secondary tab is chosen, then reset current secondary tab and change page *)

		IF( t.Tabs.PrimaryTabArray[t.Tabs.CurrentPrimaryTab].SecondaryTabArray[ss].ChangeToSecondaryTab )THEN

			//t.Tabs.PrimaryTabArray[t.Tabs.CurrentPrimaryTab].SecondaryTabArray[ss].ChangeToSecondaryTab:=	0;

			(* Change to the correct secondary tab if it has a valid PageIndex and you are not already there *)

			IF( 	(t.Tabs.PrimaryTabArray[t.Tabs.CurrentPrimaryTab].SecondaryTabArray[ss].PageIndex <> 0)
				AND	(t.Tabs.PrimaryTabArray[t.Tabs.CurrentPrimaryTab].SecondaryTabArray[ss].PageIndex <> t.PageCurrentDP)
				)THEN

				(* Change page and reset previous secondary tab CMD (CurrentPrimaryTab.CurrentSecondaryTab) *)

				t.PageChangeDP:=	t.Tabs.PrimaryTabArray[t.Tabs.CurrentPrimaryTab].SecondaryTabArray[ss].PageIndex;

				t.Tabs.PrimaryTabArray[t.Tabs.CurrentPrimaryTab]
						.SecondaryTabArray[t.Tabs.PrimaryTabArray[t.Tabs.CurrentPrimaryTab].CurrentSecondaryTab]
						.ChangeToSecondaryTab:=	0;

			ELSE

				(* Error - Reset CMD and do nothing *)

				t.Tabs.PrimaryTabArray[t.Tabs.CurrentPrimaryTab].SecondaryTabArray[ss].ChangeToSecondaryTab:=	0;

			END_IF // ChangePage

			RETURN;

		END_IF // new tab CMD

	END_IF // not CurrentSecondaryTab

END_FOR

(****************************************************)
(* Clear inactive Primary Tabs' Secondary Tabs		*)
(****************************************************)

FOR p:=0 TO HMI_MAI_TABS BY 1 DO

	(* Do not check the CurrentPrimaryTab *)

	IF( p <> t.Tabs.CurrentPrimaryTab )THEN

		FOR ss:=0 TO HMI_MAI_TABS BY 1 DO

			(* Clear ChangeToSecondaryTab *)

			t.Tabs.PrimaryTabArray[p].SecondaryTabArray[ss].ChangeToSecondaryTab:=	0;

		END_FOR (* Secondary tabs *)

	END_IF (* not current Primary *)

END_FOR (* Primary tabs *)

(****************************************************)
(* Check for 'no tab' condition						*)
(****************************************************)

(* Primary *)

PrimaryActive:=	0;

FOR p:=0 TO HMI_MAI_TABS BY 1 DO

	PrimaryActive:=	PrimaryActive OR t.Tabs.PrimaryTabArray[p].ChangeToPrimaryTab;

END_FOR

(* If no tab is active, make the current tab active *)

IF( NOT(PrimaryActive) )THEN

	t.Tabs.PrimaryTabArray[t.Tabs.CurrentPrimaryTab].ChangeToPrimaryTab:=	1;

END_IF

(* Secondary *)

SecondaryActive:=	0;

FOR ss:=0 TO HMI_MAI_TABS BY 1 DO

	SecondaryActive:=	SecondaryActive OR t.Tabs.PrimaryTabArray[t.Tabs.CurrentPrimaryTab].SecondaryTabArray[ss].ChangeToSecondaryTab;

END_FOR

(* If no tab is active, make the current tab active *)

IF( NOT(SecondaryActive) )THEN

	t.Tabs.PrimaryTabArray[t.Tabs.CurrentPrimaryTab]
			.SecondaryTabArray[t.Tabs.PrimaryTabArray[t.Tabs.CurrentPrimaryTab].CurrentSecondaryTab]
			.ChangeToSecondaryTab:=	1;

END_IF

END_FUNCTION

(* ---- HMI_Unlock.st ---- *)
(*
* File: HMI_Unlock.st
* Copyright (c) 2023 Loupe
* https://loupe.team
*
* This file is part of HMITools, licensed under the MIT License.
*
*)

(****************************************************************)
(* Unlock an item on the screen 								*)
(****************************************************************)

(* Function			DONE and TESTED DFB 20110503 *)

FUNCTION HMI_Unlock

(****************************************************************)
(* Set return value to get rid of compiler error				*)
(****************************************************************)

HMI_Unlock:=	FALSE;

(****************************************************************)
(* Set/clear proper bit in StatusDP								*)
(****************************************************************)

StatusDP.HMI_STATBIT_LOCK:=	HMI_UNLOCKED;

END_FUNCTION

(* ---- LogView.st ---- *)
(*
* File: LogView.st
* Copyright (c) 2023 Loupe
* https://loupe.team
*
* This file is part of HMITools, licensed under the MIT License.
*
*)

(* TODO: Add your comment here *)
FUNCTION LogView_init

	IF LogView.IN.CFG.MaxLogs <> 0 THEN
		BufferInit(ADR(LogView.Internal.Buffer),LogView.IN.CFG.MaxLogs,SIZEOF(LogData));
		LogView_init:=1;
	ELSE
		LogView_init:=0;
	END_IF

END_FUNCTION

FUNCTION LogView_cyclic

	LogView_cyclic:=0;

	IF NOT BufferValid(ADR(LogView.Internal.Buffer)) THEN

		LogView.OUT.STAT.Error:=1;
		LogView.OUT.STAT.ErrorID:=0;
		LogView.OUT.STAT.ErrorString:='Buffer did not initialize';

		LogView_init(LogView);
		RETURN;
	END_IF

	///////////////////////////////////////////////////////////////
	//If the logger name changes, clear the buffer and get the new
	//logger data
	///////////////////////////////////////////////////////////////

	IF LogView.Internal.LoggerName<>LogView.IN.PAR.LoggerName THEN
		LogView.Internal.LoggerName:=	LogView.IN.PAR.LoggerName;
		//Get the names of the systems logs.
		IF FIND(LogView.IN.PAR.LoggerName, 'System') <> 0 THEN
			LogView.Internal.GetIdent.Name:= '$$arlogsys'; // Double $ since it is the ST escape character
		ELSIF FIND(LogView.IN.PAR.LoggerName, 'User') <> 0 THEN
			LogView.Internal.GetIdent.Name:= '$$arlogusr';
		ELSIF FIND(LogView.IN.PAR.LoggerName, 'FieldBus') <> 0 THEN
			LogView.Internal.GetIdent.Name:= '$$fieldbus';
		ELSIF FIND(LogView.IN.PAR.LoggerName, 'Safety') <> 0 THEN
			LogView.Internal.GetIdent.Name:= '$$safety';
		ELSE
			LogView.Internal.GetIdent.Name:=LogView.IN.PAR.LoggerName;
		END_IF

	END_IF

	///////////////////////////////////////////////////////////////
	//Ensure that we always know what the top alarm is
	///////////////////////////////////////////////////////////////

	LogView.Internal.GetIdent.Execute := TRUE;
	LogView.Internal.GetIdent();
	IF LogView.Internal.GetIdent.Done THEN
		LogView.OUT.STAT.Error:=0;
		LogView.OUT.STAT.ErrorID:=0;
		LogView.OUT.STAT.ErrorString:='';
		//If this is a new ident, lets clear out the old data
		IF LogView.Internal.Ident <>  LogView.Internal.GetIdent.Ident THEN
			LogView.Internal.Ident:= LogView.Internal.GetIdent.Ident;
			BufferClear(ADR(LogView.Internal.Buffer));
		END_IF
	ELSE  (*Go to Error Step*)
		LogView.OUT.STAT.Error:=1;
		LogView.OUT.STAT.ErrorID:=LogView.Internal.GetIdent.StatusID;
		LogView.OUT.STAT.ErrorString:='Error getting log info';
		BufferClear(ADR(LogView.Internal.Buffer));
		RETURN;
	END_IF

	IF LogView.IN.CMD.GoToTop THEN
		LogView.IN.CMD.GoToTop:=0;
		LogView.IN.PAR.Offset:=0;
		LogView.Internal.OffsetIndex:=0;
	END_IF

	// Get RecordID of latest alarm
	LogView.Internal.GetRecordID.Ident := LogView.Internal.Ident;
	LogView.Internal.GetRecordID.Execute := TRUE;
	LogView.Internal.GetRecordID();
	IF LogView.Internal.GetRecordID.Error THEN
		LogView.OUT.STAT.Error:=1;
		LogView.OUT.STAT.ErrorID:=LogView.Internal.GetRecordID.StatusID;
		LogView.OUT.STAT.ErrorString:='Error getting record ID';
		BufferClear(ADR(LogView.Internal.Buffer));
		RETURN;
	END_IF

	IF LogView.IN.CMD.GoToTop THEN
		LogView.IN.CMD.GoToTop:=0;
		LogView.IN.PAR.Offset:=0;
		LogView.Internal.OffsetIndex:=0;
	END_IF
	///////////////////////////////////////////////////////////////
	//Buffer control, tells the ring buffer which way to add values
	///////////////////////////////////////////////////////////////

	//Reset offset index
	IF LogView.IN.PAR.Offset <> 0 AND LogView.Internal.OffsetIndex = 0 THEN

		//If we don't have a top, use the first alarm
		IF BufferGetItemAdr(ADR(LogView.Internal.Buffer),0,0) = 0 THEN

			LogView.Internal.OffsetIndex:=LogView.Internal.GetRecordID.RecordID;

			//If we do have a top, use the top
		ELSE

			pEntry ACCESS BufferGetItemAdr(ADR(LogView.Internal.Buffer),0,0);

			LogView.Internal.OffsetIndex:=pEntry.Index;

		END_IF
	END_IF

	//If there is an offset, the max is the offset before the offset was set
	//+- the current offset
	IF LogView.IN.PAR.Offset <> 0 OR ((LogView.Internal.OffsetIndex < LogView.Internal.GetRecordID.RecordID - 1) AND (LogView.Internal.OffsetIndex <> 0)) THEN

		//If the top value is less than or greater than where is should be in the offset
		//fill the top or bottom to allow it to get there

		MaxTopIndex:= LogView.Internal.OffsetIndex-LogView.IN.PAR.Offset;

		IF MaxTopIndex >= LogView.Internal.GetRecordID.RecordID THEN

			MaxTopIndex:=LogView.Internal.GetRecordID.RecordID;
			LogView.IN.PAR.Offset:=0;
			LogView.Internal.OffsetIndex:=LogView.Internal.GetRecordID.RecordID;

		END_IF

		//If there is no offset, fill the top
		//The bottom will fill automatically if the buffer is not full

	ELSIF LogView.IN.PAR.Offset = 0 THEN

		//Get top alarm in logger

		MaxTopIndex:=LogView.Internal.GetRecordID.RecordID;

	END_IF

	IF BufferGetItemAdr(ADR(LogView.Internal.Buffer),0,0) <> 0 THEN

		pEntry ACCESS BufferGetItemAdr(ADR(LogView.Internal.Buffer),0,0);

		IF ABS(UDINT_TO_INT(MaxTopIndex - pEntry.Index)) > UINT_TO_DINT(LogView.Internal.Buffer.MaxValues/2) THEN

			BufferClear(ADR(LogView.Internal.Buffer));

		END_IF

	END_IF

	///////////////////////////////////////////////////////////////
	//Fill the top
	///////////////////////////////////////////////////////////////

	//Fill in the top data

	IF BufferGetItemAdr(ADR(LogView.Internal.Buffer),0,0) = 0 THEN

		iNewEntry.Index:= MaxTopIndex;

		IF LogViewerGetAlarmString(LogView.Internal.GetTopAlarm,iNewEntry.Index,LogView.Internal.GetIdent.Ident,iNewEntry.String) = ERR_OK THEN

			BufferAddToTop(ADR(LogView.Internal.Buffer),ADR(iNewEntry));

		END_IF

	ELSE

		pEntry ACCESS BufferGetItemAdr(ADR(LogView.Internal.Buffer),0,0);

		iNewEntry.Index:= pEntry.Index+1;

		IF iNewEntry.Index <= MaxTopIndex THEN

			IF LogViewerGetAlarmString(LogView.Internal.GetTopAlarm, iNewEntry.Index,LogView.Internal.GetIdent.Ident,iNewEntry.String) = ERR_OK THEN

				BufferAddToTop(ADR(LogView.Internal.Buffer),ADR(iNewEntry));

			END_IF

		END_IF

	END_IF

	///////////////////////////////////////////////////////////////
	//Fill the Bottom
	///////////////////////////////////////////////////////////////

	//Get the top value to check if we should continue filling the bottom
	IF BufferGetItemAdr(ADR(LogView.Internal.Buffer),0,0) = 0 THEN

		//Do nothing let the top get one first

		//If we aren't full, OR the top index is too high, fill the bottom

	ELSIF NOT BufferFull(ADR(LogView.Internal.Buffer)) OR pEntry.Index > MaxTopIndex THEN

		//Get the last entry in the current list
		pEntry ACCESS BufferGetItemAdr(ADR(LogView.Internal.Buffer),BufferBottom(ADR(LogView.Internal.Buffer)),0);

		//Get the index lower than the last entry in the list
		iNewEntry.Index:= pEntry.Index-1;

		IF LogViewerGetAlarmString(LogView.Internal.GetBottomAlarm, iNewEntry.Index,LogView.Internal.GetIdent.Ident,iNewEntry.String) = ERR_OK THEN

			BufferAddToBottom(ADR(LogView.Internal.Buffer),ADR(iNewEntry));

		END_IF

	END_IF

	LogView.OUT.NumberAlarms:= LogView.Internal.Buffer.NumberValues;

	// These only execute on rising edge, so reset execute at end of function
	LogView.Internal.GetIdent.Execute := FALSE;
	LogView.Internal.GetIdent();
	LogView.Internal.GetRecordID.Execute := FALSE;
	LogView.Internal.GetRecordID();

END_FUNCTION

FUNCTION LogViewerCreateString

	brsmemset(ADR(emptyDTStructure), 0, SIZEOF(emptyDTStructure));
	LogViewerCreateString:=0;

	iString:='';

	IF brsmemcmp(ADR(ReadData.errTime), ADR(emptyDTStructure), SIZEOF(ReadData.errTime)) <> 0 THEN
		//Year
		IF ReadData.errTime.year<10 THEN
			brsstrcat(ADR(iString),ADR('0'));
		END_IF
		brsitoa(ReadData.errTime.year,ADR(iConvString));
		brsstrcat(ADR(iString),ADR(iConvString));
		brsstrcat(ADR(iString),ADR('-'));

		//Month
		IF ReadData.errTime.month<10 THEN
			brsstrcat(ADR(iString),ADR('0'));
		END_IF
		brsitoa(ReadData.errTime.month,ADR(iConvString));
		brsstrcat(ADR(iString),ADR(iConvString));
		brsstrcat(ADR(iString),ADR('-'));

		//Day
		IF ReadData.errTime.day<10 THEN
			brsstrcat(ADR(iString),ADR('0'));
		END_IF
		brsitoa(ReadData.errTime.day,ADR(iConvString));
		brsstrcat(ADR(iString),ADR(iConvString));

		brsstrcat(ADR(iString),ADR(' '));

		//Hour
		IF ReadData.errTime.hour<10 THEN
			brsstrcat(ADR(iString),ADR('0'));
		END_IF
		brsitoa(ReadData.errTime.hour,ADR(iConvString));
		brsstrcat(ADR(iString),ADR(iConvString));
		brsstrcat(ADR(iString),ADR(':'));

		//Minute
		IF ReadData.errTime.minute<10 THEN
			brsstrcat(ADR(iString),ADR('0'));
		END_IF
		brsitoa(ReadData.errTime.minute,ADR(iConvString));
		brsstrcat(ADR(iString),ADR(iConvString));
		brsstrcat(ADR(iString),ADR(':'));

		//Second
		IF ReadData.errTime.second<10 THEN
			brsstrcat(ADR(iString),ADR('0'));
		END_IF
		brsitoa(ReadData.errTime.second,ADR(iConvString));
		brsstrcat(ADR(iString),ADR(iConvString));
		brsstrcat(ADR(iString),ADR('.'));

		//Millisecond
		IF ReadData.errTime.millisec<100 THEN
			brsstrcat(ADR(iString),ADR('0'));
		END_IF
		IF ReadData.errTime.millisec<10 THEN
			brsstrcat(ADR(iString),ADR('0'));
		END_IF
		brsitoa(ReadData.errTime.millisec,ADR(iConvString));
		brsstrcat(ADR(iString),ADR(iConvString));
	ELSE
		brsstrcat(ADR(iString),ADR('[Invalid timestamp]'));
	END_IF

	//Error number
	brsstrcat(ADR(iString),ADR(' Err #'));
	brsitoa(ReadData.errornr,ADR(iConvString));
	brsstrcat(ADR(iString),ADR(iConvString));

	brsstrcat(ADR(iString),ADR(' '));
	brsstrcat(ADR(iString),ADR(ASCIIData));

	OutputString:= iString;

END_FUNCTION

FUNCTION LogViewerGetAlarmString

	t.ReadItem.Execute := 1;
	t.ReadItem.Ident := LoggerIdent;  (*Ident of AR logger user module from AsARLogGetIdent*)
	t.ReadItem.RecordID := recordId;
	t.ReadItem;  (* Call the Functionblock*)

	IF t.ReadItem.Done AND t.ReadItem.StatusID = 0 THEN  (*ArEventLogRead successful or last log entry read. No additional (older) entry present.*)
		t.convertUTC;
		IF t.convertUTC.status = ERR_FUB_BUSY THEN // Busy
			t.convertUTC.enable := TRUE;
			LogViewerGetAlarmString:=ERR_FUB_BUSY;
			RETURN;
		ELSIF t.convertUTC.status = ERR_FUB_ENABLE_FALSE THEN // Ready to start new conversion
			t.convertUTC.enable := TRUE;
			brsmemcpy(ADR(t.convertUTC.DT1), ADR(t.ReadItem.TimeStamp.sec), SIZEOF(t.ReadItem.TimeStamp.sec)); // DATE_AND_TIME is just a UDINT
			t.convertUTC.pDTStructure := ADR(t.ReadData.errTime);
			LogViewerGetAlarmString:=ERR_FUB_BUSY;
			RETURN;
		ELSIF t.convertUTC.status = timERR_INVALID_PARAMETER THEN
			brsmemset(ADR(t.ReadData.errTime), 0, SIZEOF(t.ReadData.errTime)); // Indicates error reading time
			t.convertUTC.enable := FALSE;
		ELSE // Done
			t.convertUTC.enable := FALSE;
			t.ReadData.errTime.millisec := UDINT_TO_UINT(t.ReadItem.TimeStamp.nsec/1000);
		END_IF

		IF t.ReadItem.AddDataFormat = arEVENTLOG_ADDFORMAT_TEXT THEN
			t.ReadAddData.Execute := 1;
			t.ReadAddData.Ident := LoggerIdent;
			t.ReadAddData.RecordID := recordId;
			t.ReadAddData.AddData := ADR(t.ASCIIData);
			t.ReadAddData.BytesToRead := SIZEOF(t.ASCIIData);
			t.ReadAddData; (* Call the function block *)
		END_IF

		LogViewerCreateString(t.ReadData,t.ASCIIData,OutputString);
		LogViewerGetAlarmString:=0;

	ELSIF t.ReadItem.StatusID = ERR_FUB_BUSY THEN

		LogViewerGetAlarmString:=ERR_FUB_BUSY;

	ELSE

		LogViewerGetAlarmString:=t.ReadItem.StatusID;

	END_IF

END_FUNCTION

(* ---- LogViewHMI.st ---- *)
(*
* File: LogViewHMI.st
* Copyright (c) 2023 Loupe
* https://loupe.team
*
* This file is part of HMITools, licensed under the MIT License.
*
*)

(* Handles displaying alarms from buffer on HMI *)
FUNCTION LogView_HMI

	//Remove warning
	LogView_HMI:=0;

	IF LogViewHMI.GoToTopButton.CMD THEN
		LogViewHMI.GoToTopButton.CMD:=0;
		LogViewHMI.internal.Offset:=0;
		LogView.IN.CMD.GoToTop:=1;
	END_IF
	IF LogViewHMI.PageUpButton.CMD THEN
		LogViewHMI.PageUpButton.CMD:=0;
		LogViewHMI.internal.Offset:=LogViewHMI.internal.Offset-10;
	END_IF
	IF LogViewHMI.PageDownButton.CMD THEN
		LogViewHMI.PageDownButton.CMD:=0;
		LogViewHMI.internal.Offset:=LogViewHMI.internal.Offset+10;
	END_IF
	IF LogViewHMI.UpButton.CMD THEN
		LogViewHMI.UpButton.CMD:=0;
		LogViewHMI.internal.Offset:=LogViewHMI.internal.Offset-1;
	END_IF
	IF LogViewHMI.DownButton.CMD THEN
		LogViewHMI.DownButton.CMD:=0;
		LogViewHMI.internal.Offset:=LogViewHMI.internal.Offset+1;
	END_IF

	LogViewHMI.internal.SelectedListIndex:= DINT_TO_UINT(LogViewHMI.ListBox.IndexDP);

	IF FIND(LogViewHMI.FilterString,'ALARM FILTER') = 1 THEN
		LogViewHMI.FilterString:='';
	END_IF

	IF LogViewHMI.internal.Offset + UDINT_TO_DINT(LogViewHMI.MaxAlarms) > UINT_TO_DINT(LogView.IN.CFG.MaxLogs) THEN
		LogView.IN.PAR.Offset:=	LogViewHMI.internal.Offset + LogViewHMI.MaxAlarms - LogView.IN.CFG.MaxLogs;
		iOffset:=				LogView.IN.CFG.MaxLogs - LogViewHMI.MaxAlarms;
		iOffsetCount:=			iOffset;
	ELSIF LogViewHMI.internal.Offset <= 0 THEN
		LogView.IN.PAR.Offset:=LogViewHMI.internal.Offset;
		iOffset:=0;
	ELSE
		LogView.IN.PAR.Offset:=1;
		iOffset:=LogViewHMI.internal.Offset-1;
	END_IF

	IF LogViewHMI.AlarmList <> 0 THEN

		pLogList ACCESS LogViewHMI.AlarmList;

		//Clear list
		brsmemset(ADR(pLogList[0]) , 0 , SIZEOF(pLogList[0]) * LogViewHMI.MaxAlarms );

		iNumDisplay:=0;

		IF LogView.OUT.STAT.Error THEN
			brsitoa(LogView.OUT.STAT.ErrorID,ADR(TempErrorID));
			TempErrorID:=CONCAT(': ',TempErrorID);
			pLogList[iNumDisplay]:= CONCAT(LogView.OUT.STAT.ErrorString,TempErrorID);
			iNumDisplay:=iNumDisplay+1;
		END_IF

		IF LogViewHMI.internal.oSelectedListIndex <> LogViewHMI.internal.SelectedListIndex AND LogViewHMI.internal.SelectedListIndex <> DINT_TO_UINT(-1) THEN
			LogViewHMI.internal.oSelectedListIndex:=-1;
		ELSE
			LogViewHMI.internal.SelectedListIndex:=-1;
		END_IF

		//Read data into array
		FOR i:=0 TO BufferBottom(ADR(LogView.Internal.Buffer)) DO

			//If there is data here, filter it and put it in the list
			IF BufferGetItemAdr(ADR(LogView.Internal.Buffer),i,0) <> 0 THEN

				//Get the next alarm
				iLogData ACCESS BufferGetItemAdr(ADR(LogView.Internal.Buffer),i,0);

				//filter data
				IF FIND(iLogData.String,LogViewHMI.FilterString) <> 0 THEN

					IF iOffset > iOffsetCount THEN
						iOffsetCount:=iOffsetCount+1;
					ELSE
						IF iNumDisplay < LogViewHMI.MaxAlarms THEN
							pLogList[iNumDisplay] := iLogData.String;

							IF LogViewHMI.internal.oSelectedListIndex = DINT_TO_UINT(-1) THEN
								IF LogViewHMI.internal.SelectedListIndex = iNumDisplay THEN
									LogViewHMI.internal.SelectedAlarmIndex:= iLogData.Index;
									LogViewHMI.internal.oSelectedListIndex:=	iNumDisplay;
									LogViewHMI.Text:=iLogData.String;
								END_IF
							ELSE
								IF LogViewHMI.internal.SelectedAlarmIndex =  iLogData.Index THEN
									LogViewHMI.internal.SelectedListIndex:=	iNumDisplay;
									LogViewHMI.Text:=iLogData.String;
								END_IF
							END_IF
							iNumDisplay:=iNumDisplay+1;
						END_IF
					END_IF
				END_IF

			ELSE

				//The last data was empty, jump out

				i:= BufferBottom(ADR(LogView.Internal.Buffer));

			END_IF

			//Limit the number of values on the diplay
			IF iNumDisplay >= LogViewHMI.MaxAlarms THEN
				i:= BufferBottom(ADR(LogView.Internal.Buffer));
			END_IF

		END_FOR

	END_IF

	LogViewHMI.internal.NumberAlarms:=iNumDisplay;

	IF brsstrcmp(ADR(LogViewHMI.FilterString),ADR('')) = 0 OR brsstrcmp(ADR(LogViewHMI.FilterString),ADR(' ')) = 0  THEN
		LogViewHMI.FilterString:='ALARM FILTER';
	END_IF

	LogViewHMI.ListBox.MaxDP:= LogViewHMI.internal.NumberAlarms;
	LogViewHMI.ListBox.MinDP:= 0;
	LogViewHMI.ListBox.IndexDP:=LogViewHMI.internal.SelectedListIndex;

END_FUNCTION

(* ---- RecipeMgr.st ---- *)
(*
* File: RecipeMgr.st
* Copyright (c) 2023 Loupe
* https://loupe.team
*
* This file is part of HMITools, licensed under the MIT License.
*
*)

(* Manage copying recipes to and from a running system and the HMI *)

FUNCTION RecipeMgr

	//**********************************************************
	// Error checking
	//**********************************************************

	IF( 	(Rec.IN.pHMIRecipe = 0)
		OR	(Rec.IN.pSystemRecipe = 0)
		OR	(Rec.IN.RecipeLength = 0)
		)THEN

		RecipeMgr:=	HMI_ERR_INVALIDINPUT;
		RETURN;

	END_IF;

	//**********************************************************
	// Handle CMDs
	//**********************************************************

	IF( Rec.HMI.RetrieveFromSystem.CMD )THEN

		// Copy from system to HMI and log
		Rec.HMI.RetrieveFromSystem.CMD:=	0;
		brsmemcpy( Rec.IN.pHMIRecipe, Rec.IN.pSystemRecipe, Rec.IN.RecipeLength );

		logInfo( Rec.IN.LoggerName, 50000, 'Recipe retrieved from system', 0 );

	END_IF;

	IF(	Rec.HMI.ApplyToSystem.CMD )THEN

		// Copy from HMI to system and log
		Rec.HMI.ApplyToSystem.CMD:=			0;
		brsmemcpy( Rec.IN.pSystemRecipe, Rec.IN.pHMIRecipe, Rec.IN.RecipeLength );

		logInfo( Rec.IN.LoggerName, 50000, 'Recipe applied to system', 0 );

	END_IF;

	IF brsmemcmp( Rec.IN.pSystemRecipe, Rec.IN.pHMIRecipe, Rec.IN.RecipeLength ) <> 0 THEN
		HMI_Show(Rec.HMI.Modified.StatusDP);
	ELSE
		HMI_Hide(Rec.HMI.Modified.StatusDP);
	END_IF

	RecipeMgr:=	HMI_ERR_OK;
	RETURN;

END_FUNCTION

(* ---- TrendFn.st ---- *)
(*
* File: TrendFn.st
* Copyright (c) 2023 Loupe
* https://loupe.team
*
* This file is part of HMITools, licensed under the MIT License.
*
*)

(************************************************************************************************************)
(* Function for controlling a trend object. Function should be called in the Init and Cyclic subroutines.	*)
(************************************************************************************************************)

(* Functionality		DONE and TESTED DFB *)

FUNCTION TrendFn

(************************************************************)
(* Set return value to get rid of compile warning 			*)
(************************************************************)

TrendFn:=	FALSE;

(************************************)
(* Call ZoomScroll FUBs 			*)
(************************************)

(* Trend *)

t.GlobalXZoomScroll();
t.GlobalYZoomScroll();

(* TimeContainer *)

t.TimeContainer.ZoomScroll();

(* ValueScale *)

FOR i:=0 TO HMI_TREND_MAI_VALUESCALE BY 1 DO

	t.ValueScale[i].ZoomScroll();

END_FOR

END_FUNCTION

(* ---- DirectoryFub.st ---- *)
(*
* File: DirectoryFub.st
* Copyright (c) 2023 Loupe
* https://loupe.team
*
* This file is part of HMITools, licensed under the MIT License.
*
*)

(*  *)
FUNCTION_BLOCK DirectoryFub

IF FileList = 0 OR Enable = 0 THEN
	Updating:=0;
	RETURN;
END_IF

Files ACCESS FileList;

	// Step through all states faster by looping 5 times
	FOR index:=0 TO 5 DO

		CASE State OF
			0:
				DirectoryRead.enable:=0;
				//CurrentFileIndex:=0; This variable is never used again.
				Updating:=1;
				State:=1;

			1:
				DirectoryOpen.enable := 	TRUE;
				DirectoryOpen.pDevice := 	ADR(FileDevice);
				DirectoryOpen.pName := 		pPath;
				DirectoryOpen();
				IF DirectoryOpen.status < ERR_FUB_ENABLE_FALSE THEN
					IF DirectoryOpen.status = ERR_OK THEN
						Ident :=			DirectoryOpen.ident;
						DirectoryOpen.enable:=	 FALSE;
						State:= 			State+1;
					ELSE
						status:= 			DirectoryOpen.status;
						State:=				10;
					END_IF;
				ELSE
					EXIT;
				END_IF;
				brsmemset(ADR(Files),0,MaxValues*(LIST_BOX_STRING_SIZE+1));
				ListFileIndex:=		0;
				status:=			ERR_FUB_BUSY;

			2:
				//read directory
				DirectoryRead.enable := 	TRUE;
				DirectoryRead.ident := 		Ident;
				DirectoryRead.pData := 		ADR(DirData);
				DirectoryRead.data_len := 	SIZEOF(DirData);
				DirectoryRead();
				IF DirectoryRead.status < ERR_FUB_ENABLE_FALSE THEN
					IF DirectoryRead.status = ERR_OK THEN
						DirectoryRead.enable := FALSE;
						State:= 			State+1;
					ELSIF DirectoryRead.status = fiERR_NO_MORE_ENTRIES THEN
						NumFiles:= 			ListFileIndex;
						status:=			ERR_OK;
						State:=				5;
					ELSE
						IF DirectoryRead.status = 20799 THEN
							status:= FileIoGetSysError();
						ELSE
							status:= DirectoryRead.status;
						END_IF;
						State:=				10;
					END_IF;
				ELSE
					EXIT;
				END_IF;

			3:
				brsstrcpy(ADR(TempString),ADR(DirData.Filename));
				iNameFilter:=NameFilter;
				//If file extension filter defined
				IF FileExt <> '' THEN
					brsmemset(ADR(TempExtension),0,SIZEOF(TempExtension));
					TempExtension:=	'.';
					brsstrcat(ADR(TempExtension),ADR(FileExt));
					//item is a File, files are filtered
					IF DirData.Mode = fiFILE THEN
						//compare just the selected extension from the file name + extension (e.g. compare ".csv" from "testing.csv")
						IF ( brsmemcmp((ADR(TempString)+(brsstrlen(ADR(TempString))-(brsstrlen(ADR(TempExtension)))))
							, ADR(TempExtension)
							, brsstrlen(ADR(TempExtension))) = 0) THEN

							//convert NameFilter to lowercase
							brsmemset(ADR(lcNameFilter),0,SIZEOF(lcNameFilter));
							FOR i:= 0 TO (SIZEOF(NameFilter) - 1) DO
								brsmemcpy(ADR(IsolatedChar),(ADR(NameFilter) + i),SIZEOF(USINT));
								IF IsolatedChar = 0 THEN// OR IsolatedChar = 46 THEN//if null or '.', dont convert file extension to lc
									EXIT;
								ELSIF IsolatedChar >=  65 AND IsolatedChar <=  90  THEN//Uppser case ascii
									brsmemset((ADR(lcNameFilter) + i),(IsolatedChar + 32),SIZEOF(USINT));
								ELSE//lower case ascii
									brsmemset((ADR(lcNameFilter) + i),IsolatedChar,SIZEOF(USINT));
								END_IF;
							END_FOR;
							//convert TempString to lowercase
							brsmemset(ADR(lcTempString),0,SIZEOF(lcTempString));
							FOR i:= 0 TO (SIZEOF(TempString) - 1) DO
								brsmemcpy(ADR(IsolatedChar),(ADR(TempString) + i),SIZEOF(USINT));
								IF IsolatedChar = 0 THEN// OR IsolatedChar = 46 THEN//if null or '.', dont convert file extension to lc
									EXIT;
								ELSIF IsolatedChar >=  65 AND IsolatedChar <=  90  THEN//Uppser case ascii
									brsmemset((ADR(lcTempString) + i),(IsolatedChar + 32),SIZEOF(USINT));
								ELSE//lower case ascii
									brsmemset((ADR(lcTempString) + i),IsolatedChar,SIZEOF(USINT));
								END_IF;
							END_FOR;
							brsmemcpy(ADR(IsolatedChar),ADR(TempString),SIZEOF(USINT));

							//Compare both lower case strings
							//Check for hidden files
							IF (FIND(lcTempString, lcNameFilter) <> 0) AND (ShowHiddenFiles OR IsolatedChar <> 46) THEN
								brsstrcpy(ADR(Files[ListFileIndex]),ADR(DirData.Filename));
								ListFileIndex:=		ListFileIndex+1;
								State:= 			State+1;
							ELSE
								State:= 			State+1;
							END_IF;

						ELSE
							State:= 			State+1;
						END_IF
					//item is a Directory, directories are not filtered
					ELSIF EnableDirectorySearch AND (brsstrcmp(ADR(DirData.Filename),ADR('.')) <> 0) THEN
						IF ((brsstrcmp(pPath,ADR('')) = 0) AND ((brsstrcmp(ADR(DirData.Filename),ADR('..')) = 0))) THEN
							State:=				State+1;
						ELSE
							brsstrcpy(ADR(Files[ListFileIndex]),ADR('\'));
							brsstrcat(ADR(Files[ListFileIndex]),ADR(DirData.Filename));
							ListFileIndex:=		ListFileIndex+1;
							State:=				State+1;
						END_IF;
					ELSE//if a directory and enabledirectorysearch is false
						State:= 				State+1;
					END_IF;
				//No extension filter defined
				ELSE
					//item is a File, files are filtered
					IF DirData.Mode = fiFILE THEN
						//convert NameFilter to lowercase
						brsmemset(ADR(lcNameFilter),0,SIZEOF(lcNameFilter));
						FOR i:= 0 TO (SIZEOF(NameFilter) - 1) DO
							brsmemcpy(ADR(IsolatedChar),(ADR(NameFilter) + i),SIZEOF(USINT));
							IF IsolatedChar = 0 THEN// OR IsolatedChar = 46 THEN//if null or '.', dont convert file extension to lc
								EXIT;
							ELSIF IsolatedChar >=  65 AND IsolatedChar <=  90  THEN//Uppser case ascii
								brsmemset((ADR(lcNameFilter) + i),(IsolatedChar + 32),SIZEOF(USINT));
							ELSE//lower case ascii
								brsmemset((ADR(lcNameFilter) + i),IsolatedChar,SIZEOF(USINT));
							END_IF;
						END_FOR;
						//convert TempString to lowercase
						brsmemset(ADR(lcTempString),0,SIZEOF(lcTempString));
						FOR i:= 0 TO (SIZEOF(TempString) - 1) DO
							brsmemcpy(ADR(IsolatedChar),(ADR(TempString) + i),SIZEOF(USINT));
							IF IsolatedChar = 0 THEN//OR IsolatedChar = 46 THEN//if null or '.', dont convert file extension to lc
								EXIT;
							ELSIF IsolatedChar >=  65 AND IsolatedChar <=  90  THEN//Uppser case ascii
								brsmemset((ADR(lcTempString) + i),(IsolatedChar + 32),SIZEOF(USINT));
							ELSE//lower case ascii
								brsmemset((ADR(lcTempString) + i),IsolatedChar,SIZEOF(USINT));
							END_IF;
						END_FOR;

						brsmemcpy(ADR(IsolatedChar),ADR(TempString),SIZEOF(USINT));

						//Compare both lower case strings
						//Check for hidden files
						IF (FIND(lcTempString, lcNameFilter) <> 0) AND (ShowHiddenFiles OR IsolatedChar <> 46) THEN
							brsstrcpy(ADR(Files[ListFileIndex]),ADR(DirData.Filename));
							ListFileIndex:=		ListFileIndex+1;
							State:= 			State+1;
						ELSE
							State:= 			State+1;
						END_IF;

					//item is a Directory, directories are not filtered
					ELSIF EnableDirectorySearch AND (brsstrcmp(ADR(DirData.Filename),ADR('.')) <> 0) THEN //item is a Directory, directories are not filtered
						IF ((brsstrcmp(pPath,ADR('')) = 0) AND ((brsstrcmp(ADR(DirData.Filename),ADR('..')) = 0))) THEN
							State:=				State+1;
						ELSE
							brsstrcpy(ADR(Files[ListFileIndex]),ADR('\'));
							brsstrcat(ADR(Files[ListFileIndex]),ADR(DirData.Filename));
							ListFileIndex:=		ListFileIndex+1;
							State:=				State+1;
						END_IF;
					ELSE//if a directory and enabledirectorysearch is false
						State:= 				State+1;
					END_IF;
				END_IF;

			4:
				IF ListFileIndex = MaxValues THEN
					status:=	ERR_OK;
					NumFiles:= 	ListFileIndex;
					State:=		5;
				ELSE
					State:=		2;
				END_IF;

			5:
				DirectoryClose.enable := 	TRUE;
				DirectoryClose.ident := 	Ident;
				DirectoryClose();
				IF DirectoryClose.status = ERR_OK THEN
					DirectoryClose.enable := FALSE;
					State:= 				6;
				END_IF;

			10:
				Initialized:=	1;
				UpdateTimer.IN:=1;
				IF UpdateTimer.Q OR iNameFilter<>NameFilter OR Refresh THEN
					Refresh:= 	0;
					State:=		0;
				END_IF

			ELSE
				Initialized:=	1;
				Updating:=		0;
				UpdateTimer.IN:=1;
				IF UpdateTimer.Q OR iNameFilter<>NameFilter OR Refresh THEN
					Refresh:= 	0;
					State:=		0;
				END_IF
		END_CASE;
	END_FOR;

UpdateTimer.PT:=T#60s;
UpdateTimer();
UpdateTimer.IN:=0;

END_FUNCTION_BLOCK

(* ---- HMI_File_Browse.st ---- *)
(*
* File: HMI_File_Browse.st
* Copyright (c) 2023 Loupe
* https://loupe.team
*
* This file is part of HMITools, licensed under the MIT License.
*
*)

FUNCTION_BLOCK HMIFileBrowse
	// Error Checks

	IF pFileList = 0 THEN
		Status :=	'Invalid entry: FileList = 0';
		RETURN;
	END_IF;

	IF MaxFiles = 0 THEN
		Status :=	'Invalid entry: MaxFiles = 0';
		RETURN;
	END_IF;

	IF pFileExtList = 0
		AND MaxExt <> 0 THEN
		Status :=	'Invalid entry: pFileExtList = 0';
		RETURN;
	END_IF;

	IF pFileExtList <> 0
		AND MaxExt = 0 THEN
		Status :=	'Invalid entry: MaxExt = 0';
		RETURN;
	END_IF;

	IF FileDevice = '' THEN
		Status :=	'Invalid entry: FileDevice = 0';
		RETURN;
	END_IF;

	IF BrowseToDirectory AND EnableDirectorySearch = FALSE THEN
		BrowseToDirectory:=	FALSE;
		Status :=	'Please enable directory search';
	END_IF;

	IF Internal.TempFileList = 0 THEN
		TMP_alloc(SIZEOF(FileSelection) * MaxFiles ,ADR(Internal.TempFileList));
	END_IF

	Internal.FileExtensionSelector.IndexDP:=FileExtIndex;
	Internal.FileExtensionSelector.Enable:=Enable;
	Internal.FileExtensionSelector.MaxDP:=MaxExt;
	Internal.FileExtensionSelector.Selection:=ADR(FileExtSelection);
	IF pFileExtList <> 0 THEN
		Internal.FileExtensionSelector.SelectionList:=pFileExtList;
	END_IF;
	Internal.FileExtensionSelector();

	Internal.Directory.Enable:=		Enable AND NOT EnableDataObjects;
	Internal.Directory.MaxValues:= 	MaxFiles;
	IF Internal.TempFileList <> 0 THEN
		Internal.Directory.FileList:=Internal.TempFileList;
	ELSE
		Internal.Directory.FileList:=pFileList;
	END_IF

	//If initial path given
	IF pDirectorySearchPath <> 0
		AND Internal.InternalBrowsingPath = '' THEN
		brsstrcpy(ADR(CurrentPath),pDirectorySearchPath);
	END_IF;

	//if command to add FileSelection to browsing path,
	IF BrowseToDirectory
		AND FileSelection <> '\..'
		AND FileSelection <> '' THEN
		BrowseToDirectory := 	FALSE;
		Refresh := 1; // do an update and navigate to directory

		//Running directory path check
		brsmemcpy(ADR(Internal.IsolatedChar),ADR(FileSelection),SIZEOF(USINT));
		IF Internal.IsolatedChar = ASCII_BACKSLASH THEN
			//add selected file to internal path
			brsstrcat(ADR(Internal.InternalBrowsingPath),(ADR(FileSelection) + 1));//Don't add first character "\" to the browsing path
			brsstrcat(ADR(Internal.InternalBrowsingPath),ADR('\'));
			//reset current path
			brsmemset(ADR(CurrentPath),0,SIZEOF(CurrentPath));
			//repopulate current path with directory path input
			IF pDirectorySearchPath <> 0 THEN
				brsstrcpy(ADR(CurrentPath),(pDirectorySearchPath));
			END_IF;
			brsstrcat(ADR(CurrentPath),ADR(Internal.InternalBrowsingPath));
			//RESET FileSelection
			FileIndex:=				-1;
			FileSelection:=			'';
		ELSE
			Status:= 				'Invalid Internal.Directory';
		END_IF;
	//If command GoToParentInternal.Directory
	ELSIF BrowseToDirectory AND FileSelection = '\..' THEN
		BrowseToDirectory :=	FALSE;
		Refresh := 1; // do an update and navigate to directory
		Internal.PathStrSize:=		UDINT_TO_UINT(brsstrlen(ADR(Internal.InternalBrowsingPath)));
		IF Internal.InternalBrowsingPath = '' THEN//at highest allowed directory, indicated by input FileDevice and Path
			Status:= 				'Invalid Internal.Directory';
		ELSE
			brsmemset(ADR(Internal.InternalBrowsingPath) +(Internal.PathStrSize - 1 ),0,SIZEOF(USINT));//remove the last character "\"
			FOR Internal.i:= 1 TO Internal.PathStrSize DO
				//isolate a single character off of the path string
				brsmemcpy(ADR(Internal.IsolatedChar),ADR(Internal.InternalBrowsingPath)+(Internal.PathStrSize-Internal.i),SIZEOF(USINT));
				//if no characters left
				IF brsstrcmp(ADR(Internal.InternalBrowsingPath),ADR('')) = 0 THEN
					EXIT;
				//if found a backslash character at the end of the string, remove it and exit
				ELSIF Internal.IsolatedChar = ASCII_BACKSLASH  THEN
					EXIT;
				//else it's a normal character, remove it
				ELSE
					brsmemset(ADR(Internal.InternalBrowsingPath) +(Internal.PathStrSize-Internal.i),0,SIZEOF(USINT));
				END_IF;
			END_FOR;
		END_IF;
		//RESET FileSelection
		FileIndex:=		-1;
		FileSelection:=	'';
		//set output to current path
		brsmemset(ADR(CurrentPath),0,SIZEOF(CurrentPath));
		IF pDirectorySearchPath <> 0 THEN
			brsstrcpy(ADR(CurrentPath),pDirectorySearchPath);
		END_IF;
		brsstrcat(ADR(CurrentPath),ADR(Internal.InternalBrowsingPath));
	ELSIF BrowseToDirectory AND FileSelection = '' THEN
		BrowseToDirectory :=	FALSE;
		Status :=	'Invalid Internal.Directory';
	END_IF;

	//If selecting a file from listbox don't update name filter
	IF FileIndex < 0 THEN
		Internal.NameFilter :=	FileSelection;
	END_IF

	//temporarly display the filter being applied
	IF FileIndex < 0 AND Internal.NameFilter <> '' THEN
		Status :=		'Filter "';
		brsstrcat(ADR(Status),ADR(Internal.NameFilter));
		brsstrcat(ADR(Status),ADR('" applied'));
	END_IF

	//Reset Internal.NameFilter if a space character is the first character
	IF (brsmemcmp(ADR(FileSelection),ADR(' '),1) = 0) THEN
		Internal.NameFilter:=		'';
		FileSelection :=	'';
		Status :=			'Name filter removed';
	END_IF

	Internal.Directory.FileExt:=		FileExtSelection;
	Internal.Directory.FileDevice:=		FileDevice;
	Internal.Directory.EnableDirectorySearch:=	EnableDirectorySearch;
	Internal.Directory.pPath:=			ADR(CurrentPath);
	Internal.Directory.NameFilter:= 	Internal.NameFilter;

	IF (Refresh) THEN
		Internal.Directory.Refresh := 1;
	END_IF

	Internal.Directory();
	Refresh := 0;

	IF EnableDataObjects AND Enable THEN
		NumFiles:= GetDataObjectList(Internal.Directory.FileList,MaxFiles);
	ELSE
		NumFiles:= 				Internal.Directory.NumFiles;
	END_IF

	IF NOT Internal.Directory.Updating
		AND Internal.TempFileList <> 0
		AND Enable
		THEN
		brsmemcpy(pFileList,Internal.TempFileList,Internal.Directory.MaxValues*(LIST_BOX_STRING_SIZE+1));
	END_IF

	//If manually changing FileSelection, reset with FileIndex to update the Internal.NameFilter
	IF Internal.oldFileSelection <> FileSelection AND FileIndex = Internal.oldFileIndex THEN
		FileIndex:=	-1;
	END_IF;

	Internal.TempFileSelection := FileSelection;

	Internal.FileNameSelector.IndexDP:=		FileIndex;
	Internal.FileNameSelector.Enable:=		Enable;
	Internal.FileNameSelector.Enable:=		TRUE;
	Internal.FileNameSelector.MaxDP:=		Internal.Directory.NumFiles;
	Internal.FileNameSelector.Selection:=	ADR(Internal.TempFileSelection);
	Internal.FileNameSelector.SelectionList:=	pFileList;
	Internal.FileNameSelector();

	//We need to read back the found index to ensure that we aren't constantly updating
	FileIndex:= Internal.FileNameSelector.IndexDP;

	FileExtIndex:=	Internal.FileExtensionSelector.IndexDP;
	//FileIndex:=Internal.oldFileSelection.IndexDP;

	IF FileIndex > -1 THEN
		FileSelection:=		Internal.TempFileSelection;
		Internal.oldFileSelection:=	FileSelection;
	END_IF;

	CompletionDP:=Internal.FileNameSelector.CompletionDP;

	//If manually changing FileSelection, reset with FileIndex to update the Internal.NameFilter
	IF Internal.oldFileSelection <> FileSelection AND FileIndex = Internal.oldFileIndex THEN
		FileIndex:=	-1;
		Internal.oldFileSelection:=	FileSelection;
	ELSE
		Internal.oldFileSelection:=	FileSelection;
	END_IF;
	IF Internal.oldFileIndex <> FileIndex THEN
		Internal.oldFileIndex:=		FileIndex;
	END_IF;

	//Reset Error String Handling
	IF Status <> '' THEN
		Internal.TON_0.IN := 	TRUE;
		Internal.TON_0.PT := 	T#2s;
		IF Internal.TON_0.Q THEN
			Internal.TON_0.IN:=	FALSE;
			brsmemset(ADR(Status),0,SIZEOF(Status));
		END_IF;
	ELSE
		Internal.TON_0.IN := 	FALSE;
	END_IF;
	Internal.TON_0();

	//If no files or directories found
	IF NumFiles = 0 AND EnableDirectorySearch = FALSE THEN
		Status:=	'No files found';
	ELSIF NumFiles = 0 AND EnableDirectorySearch = TRUE THEN
		Status:=	'No items found';
	END_IF;

END_FUNCTION_BLOCK

(* ---- HMITools.fun ---- *)
(*
* File: HMITools.fun
* Copyright (c) 2023 Loupe
* https://loupe.team
*
* This file is part of HMITools, licensed under the MIT License.
*
*)
(*
Application Ready Functions

These can be connected directly to an HMI with minimal work
*)

FUNCTION_BLOCK HMIFileBrowse (*HMI Ready file Selection function block with extensions*)
	VAR_INPUT
		Enable : BOOL; (*Enable Function Block*)
		Refresh : BOOL;
		FileDevice : STRING[80]; (*File device to look for files/directories*)
		EnableDirectorySearch : BOOL; (*Enable to look for directories*)
		EnableDataObjects : BOOL;
		BrowseToDirectory : BOOL; (*Command to browse into selected directory *)
		pDirectorySearchPath : UDINT; (*Search path within the file device*)
		pFileList : UDINT; (*List to hold file names*)
		MaxFiles : UDINT; (*Maximum number of file names list will hold*)
		pFileExtList : UDINT; (*List to hold file extensions*)
		MaxExt : UINT; (*Maximum number of file extensions list will hold*)
		FileIndex : DINT; (*Selected file index*)
		FileSelection : STRING[LIST_BOX_STRING_SIZE]; (*Selected file name*)
		FileExtIndex : DINT; (*Selected file extension index*)
		FileExtSelection : STRING[LIST_BOX_STRING_SIZE]; (*Selected file extension*)
	END_VAR
	VAR_OUTPUT
		CompletionDP : BOOL;
		CurrentPath : STRING[LIST_BOX_STRING_SIZE];
		NumFiles : UINT;
		Status : STRING[LIST_BOX_STRING_SIZE];
	END_VAR
	VAR
		Internal : HMI_File_Browse_internal_typ;
	END_VAR
END_FUNCTION_BLOCK

FUNCTION_BLOCK ListBoxFub (*HMI Ready list box*)
	VAR_INPUT
		Enable : BOOL; (*Enable function block*)
		Selection : UDINT; (*Address of Selection String*)
		SelectionList : UDINT; (*List of strings to select from*)
		IndexDP : DINT; (*List box select index*)
		MinDP : UINT; (*List box min DP*)
		MaxDP : UINT; (*List box max DP*)
		OptionDP : UINT; (*List box option DP*)
		StatusDP : UINT; (*List box Status DP*)
		ColorDP : UINT; (*List box Color DP*)
		PageSize : UINT; (*Page size*)
	END_VAR
	VAR_OUTPUT
		CompletionDP : BOOL;
	END_VAR
	VAR
		Files : REFERENCE TO ARRAY[0..0] OF STRING[LIST_BOX_STRING_SIZE];
		intIndex : DINT := 1;
		pValue : REFERENCE TO STRING[LIST_BOX_STRING_SIZE];
		oValue : STRING[LIST_BOX_STRING_SIZE];
	END_VAR
END_FUNCTION_BLOCK

FUNCTION LogView_init : BOOL (*Allocates resources for caching data from logger*)
	VAR_INPUT
		LogView : LogView_typ;
	END_VAR
END_FUNCTION

FUNCTION LogView_cyclic : BOOL (*Handles caching data from logger*)
	VAR_INPUT
		LogView : LogView_typ;
	END_VAR
	VAR
		iNewEntry : LogData;
		MaxTopIndex : UDINT;
		pEntry : REFERENCE TO LogData;
	END_VAR
END_FUNCTION

FUNCTION LogView_HMI : BOOL (*Handles displaying alarms from buffer on HMI*)
	VAR_INPUT
		LogView : LogView_typ;
		LogViewHMI : LogView_HMI_typ;
	END_VAR
	VAR
		iLogData : REFERENCE TO LogData;
		pLogList : REFERENCE TO ARRAY[0..99] OF STRING[LIST_BOX_STRING_SIZE];
		iNumDisplay : UINT;
		i : UINT;
		iOffsetCount : UDINT;
		iOffset : UDINT;
		TempErrorID : STRING[8];
	END_VAR
END_FUNCTION

FUNCTION Editor_fn : BOOL (*HMI Ready editor control *)
	VAR_INPUT
		EditorController : HMI_Editor_Controller_typ;
	END_VAR
END_FUNCTION

FUNCTION TrendFn : BOOL (*Function for controlling a trend object. Function should be called in the Init and Cyclic subroutines.*)
	VAR_IN_OUT
		t : HMI_Trend_typ; (*Trend control object*)
	END_VAR
	VAR
		i : USINT; (*Loop counter*)
	END_VAR
END_FUNCTION

FUNCTION HMI_TabControlFn_Cyclic : BOOL (*Handle tab based page switching*)
	VAR_IN_OUT
		t : HMI_Basic_typ; (*HMI_Basic control object*)
	END_VAR
	VAR
		p : UINT; (*Primary tab index*)
		ss : UINT; (*Secondary tab index for looping*)
		SecondaryTabIndex : UINT; (*Intermediate variable for primary tab page changes*)
		PrimaryActive : BOOL; (*At least one primary tab is active*)
		SecondaryActive : BOOL; (*At least one secondary tab is active*)
	END_VAR
END_FUNCTION
(*
Application Builder Functions

These functions can be used as building blocks
*)

FUNCTION HMI_Hide : BOOL (*Hide an item on the screen*)
	VAR_IN_OUT
		StatusDP : UINT; (*Item StatusDP*)
	END_VAR
END_FUNCTION

FUNCTION HMI_Show : BOOL (*Show an item on the screen*)
	VAR_IN_OUT
		StatusDP : UINT; (*Item StatusDP*)
	END_VAR
END_FUNCTION

FUNCTION HMI_Lock : BOOL (*Lock an item on the screen*)
	VAR_IN_OUT
		StatusDP : UINT; (*Item StatusDP*)
	END_VAR
END_FUNCTION

FUNCTION HMI_Unlock : BOOL (*Unlock an item on the screen*)
	VAR_IN_OUT
		StatusDP : UINT; (*Item StatusDP*)
	END_VAR
END_FUNCTION

FUNCTION HMI_SetFocus : BOOL (*Sets the focus for an item on the screen. FOCUS MUST BE RESET!*)
	VAR_IN_OUT
		StatusDP : UINT;
	END_VAR
END_FUNCTION

FUNCTION HMI_ResetFocus : BOOL (*Resets the focus bit for an item on the screen. THIS DOES NOT MOVE THE FOCUS!*)
	VAR_IN_OUT
		StatusDP : UINT;
	END_VAR
END_FUNCTION

FUNCTION HMI_OpenTouchpad : BOOL (*Opens the touchpad for an item on the screen*)
	VAR_IN_OUT
		StatusDP : UINT;
	END_VAR
END_FUNCTION

FUNCTION_BLOCK DirectoryFub (*Loads a directory and files on file extension*)
	VAR_INPUT
		Enable : BOOL; (*Enable function block*)
		Refresh : BOOL;
		EnableDirectorySearch : BOOL; (*Enable to look for directories*)
		ShowHiddenFiles : BOOL; (*Enable showing files that start with a dot*)
		FileDevice : STRING[80]; (*Directory file device*)
		pPath : UDINT; (*Search path within the file device*)
		MaxValues : UDINT; (*Maximum number of files that list will hold*)
		NameFilter : STRING[LIST_BOX_STRING_SIZE]; (*File/Diretory name filter*)
		FileList : UDINT; (*List to hold file names*)
		FileExt : STRING[LIST_BOX_STRING_SIZE]; (*File extension to filter*)
	END_VAR
	VAR_OUTPUT
		NumFiles : UINT;
		status : UINT;
		Updating : BOOL;
		Initialized : BOOL;
	END_VAR
	VAR
		DirectoryOpen : DirOpen;
		DirectoryRead : DirReadEx;
		DirectoryClose : DirClose;
		Ident : UDINT;
		State : USINT;
		ListFileIndex : UINT;
		index : UINT;
		Files : REFERENCE TO ARRAY[0..0] OF STRING[LIST_BOX_STRING_SIZE];
		DirData : fiDIR_READ_EX_DATA;
		TempString : STRING[LIST_BOX_STRING_SIZE];
		TempExtension : STRING[LIST_BOX_STRING_SIZE];
		lcTempString : STRING[LIST_BOX_STRING_SIZE];
		lcNameFilter : STRING[LIST_BOX_STRING_SIZE];
		iNameFilter : STRING[LIST_BOX_STRING_SIZE]; (*File/Diretory name filter*)
		UpdateTimer : TON;
		i : UINT;
		IsolatedChar : USINT;
	END_VAR
END_FUNCTION_BLOCK

FUNCTION EditorControl : BOOL (*Controls an HMI edit control*)
	VAR_INPUT
		Editor : HMI_EditControl_typ;
	END_VAR
END_FUNCTION

FUNCTION ControlTouch : UINT (*Handles a custom HMI control*)
	VAR_INPUT
		StatusDP : REFERENCE TO UINT;
	END_VAR
	VAR
		State : UINT;
	END_VAR
END_FUNCTION

FUNCTION ControlDismiss : BOOL (*Handles a custom HMI control*)
	VAR_INPUT
		StatusDP : REFERENCE TO UINT;
	END_VAR
END_FUNCTION

FUNCTION_BLOCK Trend_ZoomScroll (*Smart handling of trend zooming and scaling*)
	VAR_INPUT
		ZoomBase : REAL; (*Factor for zooming in and out. Will be multiplied or divided by to zoom. E.g. a ZoomBase of 2 will double or half the range when zooming in or out, respectively.*)
		ZoomIn : BOOL; (*Zoom in command*)
		ZoomOut : BOOL; (*Zoom out command*)
		ScrollBase : REAL; (*Factor for scrolling positive or negative. Percentage of current range to scroll. E.g. a ScrollBase of 0.1 will scroll 10% of current range in the positive or negative direction.*)
		ScrollPos : BOOL; (*Scroll positive command*)
		ScrollNeg : BOOL; (*Scroll negative command*)
		Reset : BOOL; (*Reset to default scroll and zoom and set to AutoUpdate scrolling*)
	END_VAR
	VAR_OUTPUT
		ZoomDP : REAL; (*ZoomDatapoint for VC object*)
		ScrollDP : REAL; (*ScrollDatapoint for VC object*)
		ModeDP : UINT; (*Mode datapoint for time scrolling (1 = AutoUpdate, 0 = No AutoUpdate).*)
	END_VAR
	VAR
		Init : BOOL; (*Flag to set ZoomDP and ScrollDP to default values*)
		Midpt : REAL; (*Current midpoint of the display. Used to calculate scroll while zooming to maintain the midpoint of the display.*)
	END_VAR
END_FUNCTION_BLOCK
(*
Log Viewer
*)

FUNCTION LogViewerGetAlarmString : UDINT
	VAR_INPUT
		t : LogView_GetAlarm;
		recordId: ArEventLogRecordIDType;
		LoggerIdent : ArEventLogIdentType;
	END_VAR
	VAR_IN_OUT
		OutputString : STRING[LIST_BOX_STRING_SIZE];
	END_VAR
END_FUNCTION

FUNCTION LogViewerCreateString : BOOL (*Log Viewer helper function to create the log string*)
	VAR_INPUT
		ReadData : ArEventLogREAD;
		ASCIIData : ARRAY[0..255] OF USINT;
	END_VAR
	VAR_IN_OUT
		OutputString : STRING[LIST_BOX_STRING_SIZE];
	END_VAR
	VAR
		iString : STRING[LIST_BOX_STRING_SIZE];
		iConvString : STRING[LIST_BOX_STRING_SIZE];
		emptyDTStructure : DTStructure;
	END_VAR
END_FUNCTION
(*
Editor Control Functions
*)

FUNCTION EditControl_CS_replaceline : UDINT (*Editor Control helper*)
	VAR_INPUT
		Text : STRING[80];
		Line : UINT;
	END_VAR
	VAR_IN_OUT
		Output : STRING[80];
	END_VAR
	VAR
		temp : STRING[80];
	END_VAR
END_FUNCTION

FUNCTION EditControl_CS_append : UDINT (*Editor Control helper*)
	VAR_INPUT
		Text : STRING[80];
	END_VAR
	VAR_IN_OUT
		Output : STRING[80];
	END_VAR
END_FUNCTION

FUNCTION EditControl_CS_getline : UDINT (*Editor Control helper *)
	VAR_INPUT
		Line : UINT;
	END_VAR
	VAR_IN_OUT
		Output : STRING[80];
	END_VAR
	VAR
		temp : STRING[80];
	END_VAR
END_FUNCTION

FUNCTION EditControl_CS_goto : UDINT (*Editor Control helper*)
	VAR_INPUT
		Line : UINT;
		Col : UINT;
	END_VAR
	VAR_IN_OUT
		Output : STRING[80];
	END_VAR
	VAR
		temp : STRING[80];
	END_VAR
END_FUNCTION

FUNCTION EditControl_CS_highlight : UDINT (*Editor Control helper*)
	VAR_INPUT
		Value : UINT;
		Mode : UINT;
	END_VAR
	VAR_IN_OUT
		Output : STRING[80];
	END_VAR
	VAR
		temp : STRING[80];
	END_VAR
END_FUNCTION

FUNCTION EditControl_CS_insert : UDINT (*Editor Control helper*)
	VAR_INPUT
		Text : STRING[80];
		Line : UINT;
	END_VAR
	VAR_IN_OUT
		Output : STRING[80];
	END_VAR
	VAR
		temp : STRING[80];
	END_VAR
END_FUNCTION

FUNCTION EditControl_CS_read : UDINT (*Editor Control helper*)
	VAR_INPUT
		Offset : UINT;
		Count : UINT;
	END_VAR
	VAR_IN_OUT
		Output : STRING[80];
	END_VAR
	VAR
		temp : STRING[80];
	END_VAR
END_FUNCTION

FUNCTION EditControl_CS_replacemarked : UDINT (*Editor Control helper*)
	VAR_INPUT
		Text : STRING[80];
	END_VAR
	VAR_IN_OUT
		Output : STRING[80];
	END_VAR
END_FUNCTION
(*
Internal Functions, these functions should not be use, they are meant only for internal use
*)

FUNCTION HMI_FindCurrentTab : BOOL (*Function to find the current primary and secondary tab based on the current page*)
	VAR_IN_OUT
		t : HMI_Basic_typ; (*HMI_Basic control object*)
	END_VAR
	VAR
		p : UINT; (*Primary tab index*)
		ss : UINT; (*Secondary tab index*)
	END_VAR
END_FUNCTION

FUNCTION FindIndexOfString : DINT (*TODO: Add your comment here*)
	VAR_INPUT
		Value : STRING[LIST_BOX_STRING_SIZE];
		List : UDINT;
		MaxList : UDINT;
	END_VAR
	VAR
		Files : REFERENCE TO ARRAY[0..0] OF STRING[LIST_BOX_STRING_SIZE];
		iteration : UDINT;
		TempString : STRING[320];
		TempString1 : STRING[320];
	END_VAR
END_FUNCTION

FUNCTION RecipeMgr : DINT (*Manage copying recipes to and from a running system and the HMI*) (*$GROUP=User*)
	VAR_INPUT
		Rec : RecipeMgr_typ;
	END_VAR
END_FUNCTION

FUNCTION_BLOCK FileQueue
	VAR_INPUT
		FileDevice : STRING[80];
		Path : STRING[320]; (*Maximum number of files that list will hold*)
		Next : BOOL;
		Cancel : BOOL;
	END_VAR
	VAR_OUTPUT
		FileName : STRING[80];
		Execute : BOOL;
		Done : BOOL;
		Busy : BOOL;
		Error : BOOL;
		ErrorID : UDINT;
	END_VAR
	VAR
		internal : RecipeUpdater_Internal_typ;
	END_VAR
END_FUNCTION_BLOCK

FUNCTION GetDataObjectList : UINT (* *) (*$GROUP=User,$CAT=User,$GROUPICON=User.png,$CATICON=User.png*)
	VAR_INPUT
		List : UDINT;
		MaxObjects : UDINT;
	END_VAR
	VAR
		Files : REFERENCE TO ARRAY[0..0] OF STRING[LIST_BOX_STRING_SIZE];
		index : UINT;
		numberVariables : UINT;
		objectIndex : UINT;
		Item : MO_List_typ;
		duplicate : BOOL;
	END_VAR
END_FUNCTION

(* ---- ListSelection.st ---- *)
(*
* File: ListSelection.st
* Copyright (c) 2023 Loupe
* https://loupe.team
*
* This file is part of HMITools, licensed under the MIT License.
*
*)

(* HMI Ready list box *)
FUNCTION_BLOCK ListBoxFub

	Files ACCESS SelectionList;
	pValue ACCESS Selection;

	MinDP:=MinDP;
	OptionDP:=OptionDP;
	StatusDP:=StatusDP;
	ColorDP:=ColorDP;
	PageSize:=PageSize;

	IF Selection = 0 OR SelectionList = 0 OR Enable = 0 THEN
		IndexDP:=intIndex:=-1;//Set index to -1 to ensure that when enable is true, it updates selection.
		RETURN;
	END_IF

	CompletionDP:=0;

	IF pValue<>oValue THEN

		intIndex:=FindIndexOfString(pValue,ADR(Files[0]),MaxDP);
		IF intIndex>=0 THEN
			IndexDP:=intIndex;
			pValue:= Files[intIndex];
			oValue:=pValue;
			CompletionDP:=1;
		ELSIF IndexDP >=0 THEN
			intIndex:=IndexDP;
			pValue:= Files[intIndex];
			oValue:=pValue;
			CompletionDP:=1;
		END_IF

	ELSIF IndexDP<>intIndex THEN

		intIndex:=IndexDP;
		pValue:= Files[intIndex];
		oValue:=pValue;
		CompletionDP:=1;

	ELSIF pValue <> Files[IndexDP] THEN

		intIndex:=FindIndexOfString(pValue,ADR(Files[0]),MaxDP);
		IndexDP:=intIndex;
		IF intIndex>=0 THEN
			pValue:= Files[intIndex];
			oValue:=pValue;
			CompletionDP:=1;
		END_IF

	END_IF;

END_FUNCTION_BLOCK

FUNCTION FindIndexOfString

	Files ACCESS List;

	FindIndexOfString:=-1;

	FOR iteration:=0 TO MaxList DO

		IF Value=''
			OR (Files[iteration] = '' AND iteration>0)
			THEN
			iteration:= MaxList;
		ELSE
			TempString:=	Files[iteration];
			TempString1:=	Value;
			ToLower(ADR(TempString));
			ToLower(ADR(TempString1));

			IF brsstrcmp(ADR(TempString),ADR(TempString1)) = 0 THEN
				FindIndexOfString:=iteration;
				iteration:= MaxList;
			END_IF
		END_IF
	END_FOR;

END_FUNCTION

(* ---- Trend_ZoomScroll.st ---- *)
(*
* File: Trend_ZoomScroll.st
* Copyright (c) 2023 Loupe
* https://loupe.team
*
* This file is part of HMITools, licensed under the MIT License.
*
*)

(********************************************************************)
(* Smart handling of trend zooming and scaling 						*)
(********************************************************************)

(* Functionality			DONE and TESTED DFB *)

FUNCTION_BLOCK Trend_ZoomScroll

	(* Initialize values on startup *)

	IF( NOT(Init) )THEN

 		Init:=	1;
		Reset:=	1;

	END_IF

	(* Reset *)

	IF( Reset )THEN

 		Reset:=		0;

		ZoomDP:=	1;
		ScrollDP:=	0;
		ModeDP:=	1;

	END_IF

	(* Zoom *)

	(* Check ZoomBase *)

	IF( ZoomBase < 1 )THEN

		(* If ZoomBase is less than 1, this will cause problems.
			Default to a ZoomBase of 1. This cancels out all Zooming *)

 		ZoomBase:=	1;

	END_IF

	IF( ZoomIn )THEN

 		ZoomIn:=	0;

		Midpt:=		ScrollDP + (0.5 / ZoomDP);	(* Midpt is ScrollDP (StartPt_curr) + Range_curr/2; Range_curr is 1/ZoomDP_curr *)
		ZoomDP:=	ZoomDP * ZoomBase; 			(* Zoom is increased by ZoomBase *)
		ScrollDP:=	Midpt - (0.5 / ZoomDP);		(* New Scroll is Midpt - Range_new/2; Range_new is 1/ZoomDP_new *)

	END_IF

	IF( ZoomOut )THEN

 		ZoomOut:=	0;

		Midpt:=		ScrollDP + (0.5 / ZoomDP);	(* Midpt is ScrollDP (StartPt_curr) + Range_curr/2; Range_curr is 1/ZoomDP_curr *)
		ZoomDP:=	ZoomDP / ZoomBase; 			(* Zoom is decreased by ZoomBase *)
		ScrollDP:=	Midpt - (0.5 / ZoomDP);		(* New Scroll is Midpt - Range_new/2; Range_new is 1/ZoomDP_new *)

	END_IF

	(* Scroll *)

	(* Check ScrollBase *)

	IF( ScrollBase < 0 )THEN

		(* If ScrollBase is less than 0, this will cause problems.
			Default to a ScrollBase of 0. This cancels out all Scrolling *)

 		ScrollBase:=	0;

	END_IF

	IF( ScrollNeg )THEN

 		ScrollNeg:=	0;

		ScrollDP:=	ScrollDP - ScrollBase / ZoomDP;	(* Decrease ScrollDP by percentage (ScrollBase) of Range. Range is 1/ZoomDP *)

	END_IF

	IF( ScrollPos )THEN

 		ScrollPos:=	0;

		ScrollDP:=	ScrollDP + ScrollBase / ZoomDP; (* Increase ScrollDP by percentage (ScrollBase) of Range. Range is 1/ZoomDP *)

	END_IF

END_FUNCTION_BLOCK

(* ---- UpdateFiles.st ---- *)
(*
* File: UpdateFiles.st
* Copyright (c) 2023 Loupe
* https://loupe.team
*
* This file is part of HMITools, licensed under the MIT License.
*
*)

(* TODO: Add your comment here *)
FUNCTION_BLOCK FileQueue

	CASE internal.State OF

		RecipeUpdater_ST_IDLE:
			Busy := FALSE;
			IF Next THEN
				Busy:=	TRUE;
				internal.DirRead.entry:= 0;
				internal.State:= RecipeUpdater_ST_ReadDirectory;
			END_IF

		RecipeUpdater_ST_ReadDirectory:

			IF internal.DirRead.status = 0 THEN
				internal.DirRead.enable:= FALSE;
				IF internal.CurrentFile.Filename[0] <> 46 THEN
					internal.State:= RecipeUpdater_ST_ReadFile;
					brsstrcpy(ADR(FileName),ADR(internal.CurrentFile.Filename));
				ELSE
					internal.DirRead.entry:= internal.DirRead.entry+1;
				END_IF
			ELSIF internal.DirRead.status = ERR_FUB_BUSY
				OR internal.DirRead.status = ERR_FUB_ENABLE_FALSE
				THEN
				internal.DirRead.enable:= TRUE;
			ELSIF internal.DirRead.status = fiERR_NO_MORE_ENTRIES
				THEN
				internal.State:= RecipeUpdater_ST_Done;
			ELSE
				Error:=	TRUE;
				ErrorID:=	internal.DirRead.status;
				internal.State:= RecipeUpdater_ST_Done;
			END_IF

		RecipeUpdater_ST_ReadFile:

			Execute:=	TRUE;
			IF NOT Next THEN
				Execute:=	FALSE;
				internal.State:= RecipeUpdater_ST_WAIT;
			ELSIF Cancel THEN
				Execute:=	FALSE;
				internal.State:= RecipeUpdater_ST_Done;
			END_IF

		RecipeUpdater_ST_WAIT:

			Execute:=	FALSE;
			IF Next THEN
				internal.State:= RecipeUpdater_ST_ReadDirectory;
				internal.DirRead.entry:= internal.DirRead.entry+1;
			ELSIF Cancel THEN
				Execute:=	FALSE;
				internal.State:= RecipeUpdater_ST_Done;
			END_IF

		RecipeUpdater_ST_Done:

			Done:= TRUE;
			Busy:=0;

			IF NOT Next
				AND NOT Cancel
				THEN
				Error:=0;
				Done:=0;
				ErrorID:=0;
				internal.State:= RecipeUpdater_ST_IDLE;
			END_IF

		RecipeUpdater_ST_:

	END_CASE

	internal.DirRead.option:=	fiFILE;
	internal.DirRead.pData:=	ADR(internal.CurrentFile);
	internal.DirRead.data_len:= SIZEOF(internal.CurrentFile);
	internal.DirRead.pDevice:=	ADR(FileDevice);
	internal.DirRead.pPath:=	ADR(Path);
	internal.DirRead();
	internal.DirRead.enable:= FALSE;

END_FUNCTION_BLOCK

(* ---- HMI_Basic.var ---- *)
(*
* File: HMI_Basic.var
* Copyright (c) 2023 Loupe
* https://loupe.team
*
* This file is part of HMITools, licensed under the MIT License.
*
*)
(*Constants*)
(*Tabs*)
VAR CONSTANT
	HMI_MAI_TABS : USINT := 9;
	HMI_INVALIDTAB : USINT := 255;
END_VAR
(*String lengths*)
VAR CONSTANT
	HMI_STRLEN_IN : UINT := 260;
	HMI_STRLEN_TIME : USINT := 9;
END_VAR
(*Locked*)
VAR CONSTANT
	HMI_UNLOCKED : BOOL := FALSE;
	HMI_LOCKED : BOOL := TRUE;
END_VAR
(*Visible*)
VAR CONSTANT
	HMI_VISIBLE : BOOL := FALSE;
	HMI_INVISIBLE : BOOL := TRUE;
END_VAR
(*Colors*)
VAR CONSTANT
	HMI_COLOR_FOREGROUND : UINT := 256;
	HMI_COLOR_BLACK : UINT := 0;
	HMI_COLOR_WHITE : UINT := 15;
	HMI_COLOR_GRAY : UINT := 7;
	HMI_COLOR_GRAY255 : UINT := 255;
	HMI_COLOR_RED : UINT := 4;
	HMI_COLOR_YELLOW : UINT := 46;
	HMI_COLOR_GREEN : UINT := 10;
END_VAR
(*Completion*)
VAR CONSTANT
	HMI_INCOMPLETE : UINT := 0;
	HMI_COMPLETE : UINT := 1;
END_VAR
(*LED values*)
VAR CONSTANT
	HMI_LED_OFF : USINT := 0;
	HMI_LED_ON : USINT := 1;
	HMI_LED_BLINKSLOW : USINT := 2;
	HMI_LED_BLINKFAST : USINT := 3;
END_VAR
(*Trend values*)
VAR CONSTANT
	HMI_TREND_MAI_CURSOR : USINT := 1;
	HMI_TREND_MAI_CURVE : USINT := 15;
	HMI_TREND_MAI_SCALECONTAINER : USINT := 4;
	HMI_TREND_MAI_VALUESCALE : USINT := 3;
END_VAR
(*ASCII values*)
VAR CONSTANT
	ASCII_BACKSLASH : USINT := 92;
END_VAR

(* ---- HMITools.var ---- *)
(*
* File: HMITools.var
* Copyright (c) 2023 Loupe
* https://loupe.team
*
* This file is part of HMITools, licensed under the MIT License.
*
*)
VAR CONSTANT
	LIST_BOX_STRING_SIZE : UINT := 260;
	fiEXTENSION : USINT := 3;
END_VAR
